LIN {X 783.157, Y -400.206, Z 104.35, A 0, B 90, C -0, E1 0, E2 0, E3 0, E4 0} C_DIS
LIN {X 784.381, Y -394.324, Z 104.35, A 0, B 90, C -0, E1 0, E2 0, E3 0, E4 0} C_DIS
LIN {X 784.236, Y -393.182, Z 104.35, A 0, B 90, C -0, E1 0, E2 0, E3 0, E4 0} C_DIS
LIN {X 783.116, Y -392.84, Z 104.35, A 0, B 90, C -0, E1 0, E2 0, E3 0, E4 0} C_DIS
LIN {X 777.125, Y -392.381, Z 104.35, A 0, B 90, C -0, E1 0, E2 0, E3 0, E4 0} C_DIS
LIN {X 776.023, Y -391.959, Z 104.35, A 0, B 90, C -0, E1 0, E2 0, E3 0, E4 0} C_DIS
LIN {X 775.424, Y -390.936, Z 104.35, A 0, B 90, C -0, E1 0, E2 0, E3 0, E4 0} C_DIS
LIN {X 773.544, Y -385.23, Z 104.35, A 0, B 90, C -0, E1 0, E2 0, E3 0, E4 0} C_DIS
LIN {X 772.847, Y -384.313, Z 104.35, A 0, B 90, C -0, E1 0, E2 0, E3 0, E4 0} C_DIS
LIN {X 771.706, Y -384.577, Z 104.35, A 0, B 90, C -0, E1 0, E2 0, E3 0, E4 0} C_DIS
LIN {X 767.372, Y -386.655, Z 104.35, A 0, B 90, C -0, E1 0, E2 0, E3 0, E4 0} C_DIS
LIN {X 766.095, Y -387.238, Z 105, A 0, B 90, C -0, E1 0, E2 0, E3 0, E4 0} C_DIS
LIN {X 764.935, Y -387.432, Z 105, A 0, B 90, C -0, E1 0, E2 0, E3 0, E4 0} C_DIS
LIN {X 763.905, Y -386.856, Z 105, A 0, B 90, C -0, E1 0, E2 0, E3 0, E4 0} C_DIS
LIN {X 759.412, Y -382.906, Z 105, A 0, B 90, C -0, E1 0, E2 0, E3 0, E4 0} C_DIS
LIN {X 758.351, Y -382.471, Z 105, A 0, B 90, C -0, E1 0, E2 0, E3 0, E4 0} C_DIS
LIN {X 757.504, Y -383.273, Z 105, A 0, B 90, C -0, E1 0, E2 0, E3 0, E4 0} C_DIS
LIN {X 754.164, Y -388.237, Z 105, A 0, B 90, C -0, E1 0, E2 0, E3 0, E4 0} C_DIS
LIN {X 753.257, Y -388.984, Z 105, A 0, B 90, C -0, E1 0, E2 0, E3 0, E4 0} C_DIS
LIN {X 752.077, Y -389, Z 105, A 0, B 90, C -0, E1 0, E2 0, E3 0, E4 0} C_DIS
LIN {X 746.211, Y -387.826, Z 105, A 0, B 90, C -0, E1 0, E2 0, E3 0, E4 0} C_DIS
LIN {X 745.074, Y -387.98, Z 105, A 0, B 90, C -0, E1 0, E2 0, E3 0, E4 0} C_DIS
LIN {X 744.742, Y -389.098, Z 105, A 0, B 90, C -0, E1 0, E2 0, E3 0, E4 0} C_DIS
LIN {X 744.331, Y -395.067, Z 105, A 0, B 90, C -0, E1 0, E2 0, E3 0, E4 0} C_DIS
LIN {X 743.919, Y -396.168, Z 105, A 0, B 90, C -0, E1 0, E2 0, E3 0, E4 0} C_DIS
LIN {X 742.906, Y -396.772, Z 105, A 0, B 90, C -0, E1 0, E2 0, E3 0, E4 0} C_DIS
LIN {X 737.238, Y -398.688, Z 105, A 0, B 90, C -0, E1 0, E2 0, E3 0, E4 0} C_DIS
LIN {X 736.331, Y -399.389, Z 105, A 0, B 90, C -0, E1 0, E2 0, E3 0, E4 0} C_DIS
LIN {X 736.602, Y -400.524, Z 105, A 0, B 90, C -0, E1 0, E2 0, E3 0, E4 0} C_DIS
LIN {X 739.231, Y -405.898, Z 105, A 0, B 90, C -0, E1 0, E2 0, E3 0, E4 0} C_DIS
LIN {X 739.424, Y -407.058, Z 105, A 0, B 90, C -0, E1 0, E2 0, E3 0, E4 0} C_DIS
LIN {X 738.849, Y -408.087, Z 105, A 0, B 90, C -0, E1 0, E2 0, E3 0, E4 0} C_DIS
LIN {X 734.899, Y -412.58, Z 105, A 0, B 90, C -0, E1 0, E2 0, E3 0, E4 0} C_DIS
LIN {X 734.463, Y -413.642, Z 105, A 0, B 90, C -0, E1 0, E2 0, E3 0, E4 0} C_DIS
LIN {X 735.266, Y -414.488, Z 105, A 0, B 90, C -0, E1 0, E2 0, E3 0, E4 0} C_DIS
LIN {X 740.229, Y -417.828, Z 105, A 0, B 90, C -0, E1 0, E2 0, E3 0, E4 0} C_DIS
LIN {X 740.977, Y -418.736, Z 105, A 0, B 90, C -0, E1 0, E2 0, E3 0, E4 0} C_DIS
LIN {X 740.993, Y -419.915, Z 105, A 0, B 90, C -0, E1 0, E2 0, E3 0, E4 0} C_DIS
LIN {X 739.819, Y -425.782, Z 105, A 0, B 90, C -0, E1 0, E2 0, E3 0, E4 0} C_DIS
LIN {X 739.972, Y -426.918, Z 105, A 0, B 90, C -0, E1 0, E2 0, E3 0, E4 0} C_DIS
LIN {X 741.091, Y -427.251, Z 105, A 0, B 90, C -0, E1 0, E2 0, E3 0, E4 0} C_DIS
LIN {X 747.059, Y -427.661, Z 105, A 0, B 90, C -0, E1 0, E2 0, E3 0, E4 0} C_DIS
LIN {X 748.16, Y -428.073, Z 105, A 0, B 90, C -0, E1 0, E2 0, E3 0, E4 0} C_DIS
LIN {X 748.764, Y -429.087, Z 105, A 0, B 90, C -0, E1 0, E2 0, E3 0, E4 0} C_DIS
LIN {X 750.68, Y -434.754, Z 105, A 0, B 90, C -0, E1 0, E2 0, E3 0, E4 0} C_DIS
LIN {X 751.382, Y -435.662, Z 105, A 0, B 90, C -0, E1 0, E2 0, E3 0, E4 0} C_DIS
LIN {X 752.516, Y -435.39, Z 105, A 0, B 90, C -0, E1 0, E2 0, E3 0, E4 0} C_DIS
LIN {X 757.89, Y -432.762, Z 105, A 0, B 90, C -0, E1 0, E2 0, E3 0, E4 0} C_DIS
LIN {X 759.05, Y -432.568, Z 105, A 0, B 90, C -0, E1 0, E2 0, E3 0, E4 0} C_DIS
LIN {X 760.08, Y -433.144, Z 105, A 0, B 90, C -0, E1 0, E2 0, E3 0, E4 0} C_DIS
LIN {X 764.573, Y -437.094, Z 105, A 0, B 90, C -0, E1 0, E2 0, E3 0, E4 0} C_DIS
LIN {X 765.634, Y -437.529, Z 105, A 0, B 90, C -0, E1 0, E2 0, E3 0, E4 0} C_DIS
LIN {X 766.481, Y -436.727, Z 105, A 0, B 90, C -0, E1 0, E2 0, E3 0, E4 0} C_DIS
LIN {X 769.821, Y -431.763, Z 105, A 0, B 90, C -0, E1 0, E2 0, E3 0, E4 0} C_DIS
LIN {X 770.728, Y -431.016, Z 105, A 0, B 90, C -0, E1 0, E2 0, E3 0, E4 0} C_DIS
LIN {X 771.908, Y -431, Z 105, A 0, B 90, C -0, E1 0, E2 0, E3 0, E4 0} C_DIS
LIN {X 777.774, Y -432.174, Z 105, A 0, B 90, C -0, E1 0, E2 0, E3 0, E4 0} C_DIS
LIN {X 778.911, Y -432.02, Z 105, A 0, B 90, C -0, E1 0, E2 0, E3 0, E4 0} C_DIS
LIN {X 779.243, Y -430.902, Z 105, A 0, B 90, C -0, E1 0, E2 0, E3 0, E4 0} C_DIS
LIN {X 779.654, Y -424.933, Z 105, A 0, B 90, C -0, E1 0, E2 0, E3 0, E4 0} C_DIS
LIN {X 780.066, Y -423.832, Z 105, A 0, B 90, C -0, E1 0, E2 0, E3 0, E4 0} C_DIS
LIN {X 781.079, Y -423.228, Z 105, A 0, B 90, C -0, E1 0, E2 0, E3 0, E4 0} C_DIS
LIN {X 786.747, Y -421.312, Z 105, A 0, B 90, C -0, E1 0, E2 0, E3 0, E4 0} C_DIS
LIN {X 787.654, Y -420.611, Z 105, A 0, B 90, C -0, E1 0, E2 0, E3 0, E4 0} C_DIS
LIN {X 787.383, Y -419.476, Z 105, A 0, B 90, C -0, E1 0, E2 0, E3 0, E4 0} C_DIS
LIN {X 784.754, Y -414.102, Z 105, A 0, B 90, C -0, E1 0, E2 0, E3 0, E4 0} C_DIS
LIN {X 784.561, Y -412.942, Z 105, A 0, B 90, C -0, E1 0, E2 0, E3 0, E4 0} C_DIS
LIN {X 785.136, Y -411.913, Z 105, A 0, B 90, C -0, E1 0, E2 0, E3 0, E4 0} C_DIS
LIN {X 789.086, Y -407.42, Z 105, A 0, B 90, C -0, E1 0, E2 0, E3 0, E4 0} C_DIS
LIN {X 789.522, Y -406.358, Z 105, A 0, B 90, C -0, E1 0, E2 0, E3 0, E4 0} C_DIS
LIN {X 788.719, Y -405.512, Z 105, A 0, B 90, C -0, E1 0, E2 0, E3 0, E4 0} C_DIS
LIN {X 783.756, Y -402.172, Z 105, A 0, B 90, C -0, E1 0, E2 0, E3 0, E4 0} C_DIS
LIN {X 783.008, Y -401.264, Z 105, A 0, B 90, C -0, E1 0, E2 0, E3 0, E4 0} C_DIS
LIN {X 782.992, Y -400.085, Z 105, A 0, B 90, C -0, E1 0, E2 0, E3 0, E4 0} C_DIS
LIN {X 784.166, Y -394.218, Z 105, A 0, B 90, C -0, E1 0, E2 0, E3 0, E4 0} C_DIS
LIN {X 784.013, Y -393.082, Z 105, A 0, B 90, C -0, E1 0, E2 0, E3 0, E4 0} C_DIS
LIN {X 782.894, Y -392.749, Z 105, A 0, B 90, C -0, E1 0, E2 0, E3 0, E4 0} C_DIS
LIN {X 776.926, Y -392.339, Z 105, A 0, B 90, C -0, E1 0, E2 0, E3 0, E4 0} C_DIS
LIN {X 775.825, Y -391.927, Z 105, A 0, B 90, C -0, E1 0, E2 0, E3 0, E4 0} C_DIS
LIN {X 775.221, Y -390.913, Z 105, A 0, B 90, C -0, E1 0, E2 0, E3 0, E4 0} C_DIS
LIN {X 773.305, Y -385.246, Z 105, A 0, B 90, C -0, E1 0, E2 0, E3 0, E4 0} C_DIS
LIN {X 772.603, Y -384.338, Z 105, A 0, B 90, C -0, E1 0, E2 0, E3 0, E4 0} C_DIS
LIN {X 771.469, Y -384.61, Z 105, A 0, B 90, C -0, E1 0, E2 0, E3 0, E4 0} C_DIS
LIN {X 767.169, Y -386.712, Z 105, A 0, B 90, C -0, E1 0, E2 0, E3 0, E4 0} C_DIS
LIN {X 765.903, Y -387.302, Z 105.65, A 0, B 90, C -0, E1 0, E2 0, E3 0, E4 0} C_DIS
LIN {X 764.75, Y -387.504, Z 105.65, A 0, B 90, C -0, E1 0, E2 0, E3 0, E4 0} C_DIS
LIN {X 763.72, Y -386.938, Z 105.65, A 0, B 90, C -0, E1 0, E2 0, E3 0, E4 0} C_DIS
LIN {X 759.215, Y -383.039, Z 105.65, A 0, B 90, C -0, E1 0, E2 0, E3 0, E4 0} C_DIS
LIN {X 758.155, Y -382.613, Z 105.65, A 0, B 90, C -0, E1 0, E2 0, E3 0, E4 0} C_DIS
LIN {X 757.318, Y -383.419, Z 105.65, A 0, B 90, C -0, E1 0, E2 0, E3 0, E4 0} C_DIS
LIN {X 754.03, Y -388.387, Z 105.65, A 0, B 90, C -0, E1 0, E2 0, E3 0, E4 0} C_DIS
LIN {X 753.132, Y -389.139, Z 105.65, A 0, B 90, C -0, E1 0, E2 0, E3 0, E4 0} C_DIS
LIN {X 751.958, Y -389.164, Z 105.65, A 0, B 90, C -0, E1 0, E2 0, E3 0, E4 0} C_DIS
LIN {X 746.107, Y -388.04, Z 105.65, A 0, B 90, C -0, E1 0, E2 0, E3 0, E4 0} C_DIS
LIN {X 744.976, Y -388.201, Z 105.65, A 0, B 90, C -0, E1 0, E2 0, E3 0, E4 0} C_DIS
LIN {X 744.654, Y -389.317, Z 105.65, A 0, B 90, C -0, E1 0, E2 0, E3 0, E4 0} C_DIS
LIN {X 744.29, Y -395.264, Z 105.65, A 0, B 90, C -0, E1 0, E2 0, E3 0, E4 0} C_DIS
LIN {X 743.889, Y -396.364, Z 105.65, A 0, B 90, C -0, E1 0, E2 0, E3 0, E4 0} C_DIS
LIN {X 742.884, Y -396.973, Z 105.65, A 0, B 90, C -0, E1 0, E2 0, E3 0, E4 0} C_DIS
LIN {X 737.255, Y -398.924, Z 105.65, A 0, B 90, C -0, E1 0, E2 0, E3 0, E4 0} C_DIS
LIN {X 736.356, Y -399.63, Z 105.65, A 0, B 90, C -0, E1 0, E2 0, E3 0, E4 0} C_DIS
LIN {X 736.635, Y -400.758, Z 105.65, A 0, B 90, C -0, E1 0, E2 0, E3 0, E4 0} C_DIS
LIN {X 739.294, Y -406.089, Z 105.65, A 0, B 90, C -0, E1 0, E2 0, E3 0, E4 0} C_DIS
LIN {X 739.496, Y -407.243, Z 105.65, A 0, B 90, C -0, E1 0, E2 0, E3 0, E4 0} C_DIS
LIN {X 738.93, Y -408.272, Z 105.65, A 0, B 90, C -0, E1 0, E2 0, E3 0, E4 0} C_DIS
LIN {X 735.031, Y -412.777, Z 105.65, A 0, B 90, C -0, E1 0, E2 0, E3 0, E4 0} C_DIS
LIN {X 734.606, Y -413.837, Z 105.65, A 0, B 90, C -0, E1 0, E2 0, E3 0, E4 0} C_DIS
LIN {X 735.411, Y -414.674, Z 105.65, A 0, B 90, C -0, E1 0, E2 0, E3 0, E4 0} C_DIS
LIN {X 740.38, Y -417.962, Z 105.65, A 0, B 90, C -0, E1 0, E2 0, E3 0, E4 0} C_DIS
LIN {X 741.131, Y -418.86, Z 105.65, A 0, B 90, C -0, E1 0, E2 0, E3 0, E4 0} C_DIS
LIN {X 741.156, Y -420.035, Z 105.65, A 0, B 90, C -0, E1 0, E2 0, E3 0, E4 0} C_DIS
LIN {X 740.032, Y -425.886, Z 105.65, A 0, B 90, C -0, E1 0, E2 0, E3 0, E4 0} C_DIS
LIN {X 740.193, Y -427.016, Z 105.65, A 0, B 90, C -0, E1 0, E2 0, E3 0, E4 0} C_DIS
LIN {X 741.31, Y -427.339, Z 105.65, A 0, B 90, C -0, E1 0, E2 0, E3 0, E4 0} C_DIS
LIN {X 747.256, Y -427.702, Z 105.65, A 0, B 90, C -0, E1 0, E2 0, E3 0, E4 0} C_DIS
LIN {X 748.356, Y -428.104, Z 105.65, A 0, B 90, C -0, E1 0, E2 0, E3 0, E4 0} C_DIS
LIN {X 748.965, Y -429.109, Z 105.65, A 0, B 90, C -0, E1 0, E2 0, E3 0, E4 0} C_DIS
LIN {X 750.917, Y -434.738, Z 105.65, A 0, B 90, C -0, E1 0, E2 0, E3 0, E4 0} C_DIS
LIN {X 751.622, Y -435.636, Z 105.65, A 0, B 90, C -0, E1 0, E2 0, E3 0, E4 0} C_DIS
LIN {X 752.75, Y -435.357, Z 105.65, A 0, B 90, C -0, E1 0, E2 0, E3 0, E4 0} C_DIS
LIN {X 758.082, Y -432.698, Z 105.65, A 0, B 90, C -0, E1 0, E2 0, E3 0, E4 0} C_DIS
LIN {X 759.235, Y -432.496, Z 105.65, A 0, B 90, C -0, E1 0, E2 0, E3 0, E4 0} C_DIS
LIN {X 760.265, Y -433.062, Z 105.65, A 0, B 90, C -0, E1 0, E2 0, E3 0, E4 0} C_DIS
LIN {X 764.77, Y -436.961, Z 105.65, A 0, B 90, C -0, E1 0, E2 0, E3 0, E4 0} C_DIS
LIN {X 765.83, Y -437.387, Z 105.65, A 0, B 90, C -0, E1 0, E2 0, E3 0, E4 0} C_DIS
LIN {X 766.667, Y -436.581, Z 105.65, A 0, B 90, C -0, E1 0, E2 0, E3 0, E4 0} C_DIS
LIN {X 769.955, Y -431.613, Z 105.65, A 0, B 90, C -0, E1 0, E2 0, E3 0, E4 0} C_DIS
LIN {X 770.853, Y -430.861, Z 105.65, A 0, B 90, C -0, E1 0, E2 0, E3 0, E4 0} C_DIS
LIN {X 772.027, Y -430.836, Z 105.65, A 0, B 90, C -0, E1 0, E2 0, E3 0, E4 0} C_DIS
LIN {X 777.878, Y -431.96, Z 105.65, A 0, B 90, C -0, E1 0, E2 0, E3 0, E4 0} C_DIS
LIN {X 779.009, Y -431.799, Z 105.65, A 0, B 90, C -0, E1 0, E2 0, E3 0, E4 0} C_DIS
LIN {X 779.331, Y -430.683, Z 105.65, A 0, B 90, C -0, E1 0, E2 0, E3 0, E4 0} C_DIS
LIN {X 779.695, Y -424.736, Z 105.65, A 0, B 90, C -0, E1 0, E2 0, E3 0, E4 0} C_DIS
LIN {X 780.096, Y -423.636, Z 105.65, A 0, B 90, C -0, E1 0, E2 0, E3 0, E4 0} C_DIS
LIN {X 781.101, Y -423.027, Z 105.65, A 0, B 90, C -0, E1 0, E2 0, E3 0, E4 0} C_DIS
LIN {X 786.73, Y -421.076, Z 105.65, A 0, B 90, C -0, E1 0, E2 0, E3 0, E4 0} C_DIS
LIN {X 787.629, Y -420.37, Z 105.65, A 0, B 90, C -0, E1 0, E2 0, E3 0, E4 0} C_DIS
LIN {X 787.349, Y -419.242, Z 105.65, A 0, B 90, C -0, E1 0, E2 0, E3 0, E4 0} C_DIS
LIN {X 784.691, Y -413.911, Z 105.65, A 0, B 90, C -0, E1 0, E2 0, E3 0, E4 0} C_DIS
LIN {X 784.489, Y -412.757, Z 105.65, A 0, B 90, C -0, E1 0, E2 0, E3 0, E4 0} C_DIS
LIN {X 785.055, Y -411.728, Z 105.65, A 0, B 90, C -0, E1 0, E2 0, E3 0, E4 0} C_DIS
LIN {X 788.954, Y -407.223, Z 105.65, A 0, B 90, C -0, E1 0, E2 0, E3 0, E4 0} C_DIS
LIN {X 789.379, Y -406.163, Z 105.65, A 0, B 90, C -0, E1 0, E2 0, E3 0, E4 0} C_DIS
LIN {X 788.573, Y -405.326, Z 105.65, A 0, B 90, C -0, E1 0, E2 0, E3 0, E4 0} C_DIS
LIN {X 783.605, Y -402.038, Z 105.65, A 0, B 90, C -0, E1 0, E2 0, E3 0, E4 0} C_DIS
LIN {X 782.854, Y -401.14, Z 105.65, A 0, B 90, C -0, E1 0, E2 0, E3 0, E4 0} C_DIS
LIN {X 782.829, Y -399.965, Z 105.65, A 0, B 90, C -0, E1 0, E2 0, E3 0, E4 0} C_DIS
LIN {X 783.953, Y -394.114, Z 105.65, A 0, B 90, C -0, E1 0, E2 0, E3 0, E4 0} C_DIS
LIN {X 783.791, Y -392.984, Z 105.65, A 0, B 90, C -0, E1 0, E2 0, E3 0, E4 0} C_DIS
LIN {X 782.675, Y -392.661, Z 105.65, A 0, B 90, C -0, E1 0, E2 0, E3 0, E4 0} C_DIS
LIN {X 776.728, Y -392.298, Z 105.65, A 0, B 90, C -0, E1 0, E2 0, E3 0, E4 0} C_DIS
LIN {X 775.629, Y -391.896, Z 105.65, A 0, B 90, C -0, E1 0, E2 0, E3 0, E4 0} C_DIS
LIN {X 775.02, Y -390.891, Z 105.65, A 0, B 90, C -0, E1 0, E2 0, E3 0, E4 0} C_DIS
LIN {X 773.068, Y -385.262, Z 105.65, A 0, B 90, C -0, E1 0, E2 0, E3 0, E4 0} C_DIS
LIN {X 772.363, Y -384.364, Z 105.65, A 0, B 90, C -0, E1 0, E2 0, E3 0, E4 0} C_DIS
LIN {X 771.235, Y -384.643, Z 105.65, A 0, B 90, C -0, E1 0, E2 0, E3 0, E4 0} C_DIS
LIN {X 766.97, Y -386.77, Z 105.65, A 0, B 90, C -0, E1 0, E2 0, E3 0, E4 0} C_DIS
LIN {X 765.714, Y -387.365, Z 106.3, A 0, B 90, C -0, E1 0, E2 0, E3 0, E4 0} C_DIS
LIN {X 764.567, Y -387.575, Z 106.3, A 0, B 90, C -0, E1 0, E2 0, E3 0, E4 0} C_DIS
LIN {X 763.537, Y -387.02, Z 106.3, A 0, B 90, C -0, E1 0, E2 0, E3 0, E4 0} C_DIS
LIN {X 759.022, Y -383.171, Z 106.3, A 0, B 90, C -0, E1 0, E2 0, E3 0, E4 0} C_DIS
LIN {X 757.963, Y -382.755, Z 106.3, A 0, B 90, C -0, E1 0, E2 0, E3 0, E4 0} C_DIS
LIN {X 757.135, Y -383.564, Z 106.3, A 0, B 90, C -0, E1 0, E2 0, E3 0, E4 0} C_DIS
LIN {X 753.898, Y -388.537, Z 106.3, A 0, B 90, C -0, E1 0, E2 0, E3 0, E4 0} C_DIS
LIN {X 753.01, Y -389.292, Z 106.3, A 0, B 90, C -0, E1 0, E2 0, E3 0, E4 0} C_DIS
LIN {X 751.84, Y -389.326, Z 106.3, A 0, B 90, C -0, E1 0, E2 0, E3 0, E4 0} C_DIS
LIN {X 746.005, Y -388.251, Z 106.3, A 0, B 90, C -0, E1 0, E2 0, E3 0, E4 0} C_DIS
LIN {X 744.88, Y -388.42, Z 106.3, A 0, B 90, C -0, E1 0, E2 0, E3 0, E4 0} C_DIS
LIN {X 744.568, Y -389.534, Z 106.3, A 0, B 90, C -0, E1 0, E2 0, E3 0, E4 0} C_DIS
LIN {X 744.251, Y -395.459, Z 106.3, A 0, B 90, C -0, E1 0, E2 0, E3 0, E4 0} C_DIS
LIN {X 743.859, Y -396.558, Z 106.3, A 0, B 90, C -0, E1 0, E2 0, E3 0, E4 0} C_DIS
LIN {X 742.864, Y -397.172, Z 106.3, A 0, B 90, C -0, E1 0, E2 0, E3 0, E4 0} C_DIS
LIN {X 737.273, Y -399.158, Z 106.3, A 0, B 90, C -0, E1 0, E2 0, E3 0, E4 0} C_DIS
LIN {X 736.383, Y -399.867, Z 106.3, A 0, B 90, C -0, E1 0, E2 0, E3 0, E4 0} C_DIS
LIN {X 736.67, Y -400.989, Z 106.3, A 0, B 90, C -0, E1 0, E2 0, E3 0, E4 0} C_DIS
LIN {X 739.358, Y -406.278, Z 106.3, A 0, B 90, C -0, E1 0, E2 0, E3 0, E4 0} C_DIS
LIN {X 739.568, Y -407.425, Z 106.3, A 0, B 90, C -0, E1 0, E2 0, E3 0, E4 0} C_DIS
LIN {X 739.012, Y -408.455, Z 106.3, A 0, B 90, C -0, E1 0, E2 0, E3 0, E4 0} C_DIS
LIN {X 735.164, Y -412.971, Z 106.3, A 0, B 90, C -0, E1 0, E2 0, E3 0, E4 0} C_DIS
LIN {X 734.748, Y -414.03, Z 106.3, A 0, B 90, C -0, E1 0, E2 0, E3 0, E4 0} C_DIS
LIN {X 735.557, Y -414.857, Z 106.3, A 0, B 90, C -0, E1 0, E2 0, E3 0, E4 0} C_DIS
LIN {X 740.529, Y -418.094, Z 106.3, A 0, B 90, C -0, E1 0, E2 0, E3 0, E4 0} C_DIS
LIN {X 741.285, Y -418.982, Z 106.3, A 0, B 90, C -0, E1 0, E2 0, E3 0, E4 0} C_DIS
LIN {X 741.319, Y -420.152, Z 106.3, A 0, B 90, C -0, E1 0, E2 0, E3 0, E4 0} C_DIS
LIN {X 740.243, Y -425.987, Z 106.3, A 0, B 90, C -0, E1 0, E2 0, E3 0, E4 0} C_DIS
LIN {X 740.413, Y -427.112, Z 106.3, A 0, B 90, C -0, E1 0, E2 0, E3 0, E4 0} C_DIS
LIN {X 741.527, Y -427.425, Z 106.3, A 0, B 90, C -0, E1 0, E2 0, E3 0, E4 0} C_DIS
LIN {X 747.452, Y -427.741, Z 106.3, A 0, B 90, C -0, E1 0, E2 0, E3 0, E4 0} C_DIS
LIN {X 748.55, Y -428.133, Z 106.3, A 0, B 90, C -0, E1 0, E2 0, E3 0, E4 0} C_DIS
LIN {X 749.164, Y -429.129, Z 106.3, A 0, B 90, C -0, E1 0, E2 0, E3 0, E4 0} C_DIS
LIN {X 751.151, Y -434.72, Z 106.3, A 0, B 90, C -0, E1 0, E2 0, E3 0, E4 0} C_DIS
LIN {X 751.86, Y -435.609, Z 106.3, A 0, B 90, C -0, E1 0, E2 0, E3 0, E4 0} C_DIS
LIN {X 752.981, Y -435.323, Z 106.3, A 0, B 90, C -0, E1 0, E2 0, E3 0, E4 0} C_DIS
LIN {X 758.271, Y -432.635, Z 106.3, A 0, B 90, C -0, E1 0, E2 0, E3 0, E4 0} C_DIS
LIN {X 759.418, Y -432.425, Z 106.3, A 0, B 90, C -0, E1 0, E2 0, E3 0, E4 0} C_DIS
LIN {X 760.447, Y -432.98, Z 106.3, A 0, B 90, C -0, E1 0, E2 0, E3 0, E4 0} C_DIS
LIN {X 764.963, Y -436.829, Z 106.3, A 0, B 90, C -0, E1 0, E2 0, E3 0, E4 0} C_DIS
LIN {X 766.022, Y -437.245, Z 106.3, A 0, B 90, C -0, E1 0, E2 0, E3 0, E4 0} C_DIS
LIN {X 766.85, Y -436.436, Z 106.3, A 0, B 90, C -0, E1 0, E2 0, E3 0, E4 0} C_DIS
LIN {X 770.087, Y -431.463, Z 106.3, A 0, B 90, C -0, E1 0, E2 0, E3 0, E4 0} C_DIS
LIN {X 770.975, Y -430.708, Z 106.3, A 0, B 90, C -0, E1 0, E2 0, E3 0, E4 0} C_DIS
LIN {X 772.145, Y -430.674, Z 106.3, A 0, B 90, C -0, E1 0, E2 0, E3 0, E4 0} C_DIS
LIN {X 777.98, Y -431.749, Z 106.3, A 0, B 90, C -0, E1 0, E2 0, E3 0, E4 0} C_DIS
LIN {X 779.105, Y -431.58, Z 106.3, A 0, B 90, C -0, E1 0, E2 0, E3 0, E4 0} C_DIS
LIN {X 779.417, Y -430.466, Z 106.3, A 0, B 90, C -0, E1 0, E2 0, E3 0, E4 0} C_DIS
LIN {X 779.734, Y -424.541, Z 106.3, A 0, B 90, C -0, E1 0, E2 0, E3 0, E4 0} C_DIS
LIN {X 780.125, Y -423.442, Z 106.3, A 0, B 90, C -0, E1 0, E2 0, E3 0, E4 0} C_DIS
LIN {X 781.121, Y -422.828, Z 106.3, A 0, B 90, C -0, E1 0, E2 0, E3 0, E4 0} C_DIS
LIN {X 786.712, Y -420.842, Z 106.3, A 0, B 90, C -0, E1 0, E2 0, E3 0, E4 0} C_DIS
LIN {X 787.602, Y -420.133, Z 106.3, A 0, B 90, C -0, E1 0, E2 0, E3 0, E4 0} C_DIS
LIN {X 787.315, Y -419.011, Z 106.3, A 0, B 90, C -0, E1 0, E2 0, E3 0, E4 0} C_DIS
LIN {X 784.627, Y -413.722, Z 106.3, A 0, B 90, C -0, E1 0, E2 0, E3 0, E4 0} C_DIS
LIN {X 784.417, Y -412.575, Z 106.3, A 0, B 90, C -0, E1 0, E2 0, E3 0, E4 0} C_DIS
LIN {X 784.973, Y -411.545, Z 106.3, A 0, B 90, C -0, E1 0, E2 0, E3 0, E4 0} C_DIS
LIN {X 788.821, Y -407.029, Z 106.3, A 0, B 90, C -0, E1 0, E2 0, E3 0, E4 0} C_DIS
LIN {X 789.237, Y -405.97, Z 106.3, A 0, B 90, C -0, E1 0, E2 0, E3 0, E4 0} C_DIS
LIN {X 788.428, Y -405.143, Z 106.3, A 0, B 90, C -0, E1 0, E2 0, E3 0, E4 0} C_DIS
LIN {X 783.456, Y -401.906, Z 106.3, A 0, B 90, C -0, E1 0, E2 0, E3 0, E4 0} C_DIS
LIN {X 782.7, Y -401.018, Z 106.3, A 0, B 90, C -0, E1 0, E2 0, E3 0, E4 0} C_DIS
LIN {X 782.666, Y -399.848, Z 106.3, A 0, B 90, C -0, E1 0, E2 0, E3 0, E4 0} C_DIS
LIN {X 783.742, Y -394.013, Z 106.3, A 0, B 90, C -0, E1 0, E2 0, E3 0, E4 0} C_DIS
LIN {X 783.572, Y -392.888, Z 106.3, A 0, B 90, C -0, E1 0, E2 0, E3 0, E4 0} C_DIS
LIN {X 782.458, Y -392.575, Z 106.3, A 0, B 90, C -0, E1 0, E2 0, E3 0, E4 0} C_DIS
LIN {X 776.533, Y -392.259, Z 106.3, A 0, B 90, C -0, E1 0, E2 0, E3 0, E4 0} C_DIS
LIN {X 775.435, Y -391.867, Z 106.3, A 0, B 90, C -0, E1 0, E2 0, E3 0, E4 0} C_DIS
LIN {X 774.821, Y -390.871, Z 106.3, A 0, B 90, C -0, E1 0, E2 0, E3 0, E4 0} C_DIS
LIN {X 772.834, Y -385.28, Z 106.3, A 0, B 90, C -0, E1 0, E2 0, E3 0, E4 0} C_DIS
LIN {X 772.125, Y -384.391, Z 106.3, A 0, B 90, C -0, E1 0, E2 0, E3 0, E4 0} C_DIS
LIN {X 771.004, Y -384.677, Z 106.3, A 0, B 90, C -0, E1 0, E2 0, E3 0, E4 0} C_DIS
LIN {X 766.772, Y -386.828, Z 106.3, A 0, B 90, C -0, E1 0, E2 0, E3 0, E4 0} C_DIS
LIN {X 765.528, Y -387.429, Z 106.95, A 0, B 90, C -0, E1 0, E2 0, E3 0, E4 0} C_DIS
LIN {X 764.387, Y -387.647, Z 106.95, A 0, B 90, C -0, E1 0, E2 0, E3 0, E4 0} C_DIS
LIN {X 763.357, Y -387.102, Z 106.95, A 0, B 90, C -0, E1 0, E2 0, E3 0, E4 0} C_DIS
LIN {X 758.831, Y -383.303, Z 106.95, A 0, B 90, C -0, E1 0, E2 0, E3 0, E4 0} C_DIS
LIN {X 757.773, Y -382.897, Z 106.95, A 0, B 90, C -0, E1 0, E2 0, E3 0, E4 0} C_DIS
LIN {X 756.955, Y -383.708, Z 106.95, A 0, B 90, C -0, E1 0, E2 0, E3 0, E4 0} C_DIS
LIN {X 753.769, Y -388.685, Z 106.95, A 0, B 90, C -0, E1 0, E2 0, E3 0, E4 0} C_DIS
LIN {X 752.89, Y -389.444, Z 106.95, A 0, B 90, C -0, E1 0, E2 0, E3 0, E4 0} C_DIS
LIN {X 751.725, Y -389.487, Z 106.95, A 0, B 90, C -0, E1 0, E2 0, E3 0, E4 0} C_DIS
LIN {X 745.906, Y -388.46, Z 106.95, A 0, B 90, C -0, E1 0, E2 0, E3 0, E4 0} C_DIS
LIN {X 744.787, Y -388.637, Z 106.95, A 0, B 90, C -0, E1 0, E2 0, E3 0, E4 0} C_DIS
LIN {X 744.484, Y -389.749, Z 106.95, A 0, B 90, C -0, E1 0, E2 0, E3 0, E4 0} C_DIS
LIN {X 744.213, Y -395.653, Z 106.95, A 0, B 90, C -0, E1 0, E2 0, E3 0, E4 0} C_DIS
LIN {X 743.832, Y -396.749, Z 106.95, A 0, B 90, C -0, E1 0, E2 0, E3 0, E4 0} C_DIS
LIN {X 742.844, Y -397.369, Z 106.95, A 0, B 90, C -0, E1 0, E2 0, E3 0, E4 0} C_DIS
LIN {X 737.291, Y -399.389, Z 106.95, A 0, B 90, C -0, E1 0, E2 0, E3 0, E4 0} C_DIS
LIN {X 736.411, Y -400.102, Z 106.95, A 0, B 90, C -0, E1 0, E2 0, E3 0, E4 0} C_DIS
LIN {X 736.704, Y -401.217, Z 106.95, A 0, B 90, C -0, E1 0, E2 0, E3 0, E4 0} C_DIS
LIN {X 739.422, Y -406.464, Z 106.95, A 0, B 90, C -0, E1 0, E2 0, E3 0, E4 0} C_DIS
LIN {X 739.639, Y -407.605, Z 106.95, A 0, B 90, C -0, E1 0, E2 0, E3 0, E4 0} C_DIS
LIN {X 739.094, Y -408.635, Z 106.95, A 0, B 90, C -0, E1 0, E2 0, E3 0, E4 0} C_DIS
LIN {X 735.295, Y -413.162, Z 106.95, A 0, B 90, C -0, E1 0, E2 0, E3 0, E4 0} C_DIS
LIN {X 734.889, Y -414.219, Z 106.95, A 0, B 90, C -0, E1 0, E2 0, E3 0, E4 0} C_DIS
LIN {X 735.701, Y -415.038, Z 106.95, A 0, B 90, C -0, E1 0, E2 0, E3 0, E4 0} C_DIS
LIN {X 740.678, Y -418.224, Z 106.95, A 0, B 90, C -0, E1 0, E2 0, E3 0, E4 0} C_DIS
LIN {X 741.437, Y -419.103, Z 106.95, A 0, B 90, C -0, E1 0, E2 0, E3 0, E4 0} C_DIS
LIN {X 741.479, Y -420.267, Z 106.95, A 0, B 90, C -0, E1 0, E2 0, E3 0, E4 0} C_DIS
LIN {X 740.453, Y -426.087, Z 106.95, A 0, B 90, C -0, E1 0, E2 0, E3 0, E4 0} C_DIS
LIN {X 740.63, Y -427.206, Z 106.95, A 0, B 90, C -0, E1 0, E2 0, E3 0, E4 0} C_DIS
LIN {X 741.742, Y -427.509, Z 106.95, A 0, B 90, C -0, E1 0, E2 0, E3 0, E4 0} C_DIS
LIN {X 747.645, Y -427.779, Z 106.95, A 0, B 90, C -0, E1 0, E2 0, E3 0, E4 0} C_DIS
LIN {X 748.742, Y -428.161, Z 106.95, A 0, B 90, C -0, E1 0, E2 0, E3 0, E4 0} C_DIS
LIN {X 749.361, Y -429.148, Z 106.95, A 0, B 90, C -0, E1 0, E2 0, E3 0, E4 0} C_DIS
LIN {X 751.382, Y -434.701, Z 106.95, A 0, B 90, C -0, E1 0, E2 0, E3 0, E4 0} C_DIS
LIN {X 752.095, Y -435.582, Z 106.95, A 0, B 90, C -0, E1 0, E2 0, E3 0, E4 0} C_DIS
LIN {X 753.209, Y -435.288, Z 106.95, A 0, B 90, C -0, E1 0, E2 0, E3 0, E4 0} C_DIS
LIN {X 758.457, Y -432.571, Z 106.95, A 0, B 90, C -0, E1 0, E2 0, E3 0, E4 0} C_DIS
LIN {X 759.598, Y -432.353, Z 106.95, A 0, B 90, C -0, E1 0, E2 0, E3 0, E4 0} C_DIS
LIN {X 760.628, Y -432.898, Z 106.95, A 0, B 90, C -0, E1 0, E2 0, E3 0, E4 0} C_DIS
LIN {X 765.154, Y -436.697, Z 106.95, A 0, B 90, C -0, E1 0, E2 0, E3 0, E4 0} C_DIS
LIN {X 766.212, Y -437.103, Z 106.95, A 0, B 90, C -0, E1 0, E2 0, E3 0, E4 0} C_DIS
LIN {X 767.03, Y -436.292, Z 106.95, A 0, B 90, C -0, E1 0, E2 0, E3 0, E4 0} C_DIS
LIN {X 770.216, Y -431.315, Z 106.95, A 0, B 90, C -0, E1 0, E2 0, E3 0, E4 0} C_DIS
LIN {X 771.095, Y -430.556, Z 106.95, A 0, B 90, C -0, E1 0, E2 0, E3 0, E4 0} C_DIS
LIN {X 772.26, Y -430.513, Z 106.95, A 0, B 90, C -0, E1 0, E2 0, E3 0, E4 0} C_DIS
LIN {X 778.079, Y -431.54, Z 106.95, A 0, B 90, C -0, E1 0, E2 0, E3 0, E4 0} C_DIS
LIN {X 779.198, Y -431.363, Z 106.95, A 0, B 90, C -0, E1 0, E2 0, E3 0, E4 0} C_DIS
LIN {X 779.501, Y -430.251, Z 106.95, A 0, B 90, C -0, E1 0, E2 0, E3 0, E4 0} C_DIS
LIN {X 779.772, Y -424.347, Z 106.95, A 0, B 90, C -0, E1 0, E2 0, E3 0, E4 0} C_DIS
LIN {X 780.153, Y -423.251, Z 106.95, A 0, B 90, C -0, E1 0, E2 0, E3 0, E4 0} C_DIS
LIN {X 781.141, Y -422.631, Z 106.95, A 0, B 90, C -0, E1 0, E2 0, E3 0, E4 0} C_DIS
LIN {X 786.694, Y -420.611, Z 106.95, A 0, B 90, C -0, E1 0, E2 0, E3 0, E4 0} C_DIS
LIN {X 787.574, Y -419.898, Z 106.95, A 0, B 90, C -0, E1 0, E2 0, E3 0, E4 0} C_DIS
LIN {X 787.281, Y -418.783, Z 106.95, A 0, B 90, C -0, E1 0, E2 0, E3 0, E4 0} C_DIS
LIN {X 784.563, Y -413.536, Z 106.95, A 0, B 90, C -0, E1 0, E2 0, E3 0, E4 0} C_DIS
LIN {X 784.346, Y -412.395, Z 106.95, A 0, B 90, C -0, E1 0, E2 0, E3 0, E4 0} C_DIS
LIN {X 784.891, Y -411.365, Z 106.95, A 0, B 90, C -0, E1 0, E2 0, E3 0, E4 0} C_DIS
LIN {X 788.69, Y -406.838, Z 106.95, A 0, B 90, C -0, E1 0, E2 0, E3 0, E4 0} C_DIS
LIN {X 789.096, Y -405.781, Z 106.95, A 0, B 90, C -0, E1 0, E2 0, E3 0, E4 0} C_DIS
LIN {X 788.284, Y -404.962, Z 106.95, A 0, B 90, C -0, E1 0, E2 0, E3 0, E4 0} C_DIS
LIN {X 783.307, Y -401.776, Z 106.95, A 0, B 90, C -0, E1 0, E2 0, E3 0, E4 0} C_DIS
LIN {X 782.548, Y -400.897, Z 106.95, A 0, B 90, C -0, E1 0, E2 0, E3 0, E4 0} C_DIS
LIN {X 782.506, Y -399.733, Z 106.95, A 0, B 90, C -0, E1 0, E2 0, E3 0, E4 0} C_DIS
LIN {X 783.532, Y -393.913, Z 106.95, A 0, B 90, C -0, E1 0, E2 0, E3 0, E4 0} C_DIS
LIN {X 783.355, Y -392.794, Z 106.95, A 0, B 90, C -0, E1 0, E2 0, E3 0, E4 0} C_DIS
LIN {X 782.243, Y -392.491, Z 106.95, A 0, B 90, C -0, E1 0, E2 0, E3 0, E4 0} C_DIS
LIN {X 776.34, Y -392.221, Z 106.95, A 0, B 90, C -0, E1 0, E2 0, E3 0, E4 0} C_DIS
LIN {X 775.243, Y -391.839, Z 106.95, A 0, B 90, C -0, E1 0, E2 0, E3 0, E4 0} C_DIS
LIN {X 774.624, Y -390.852, Z 106.95, A 0, B 90, C -0, E1 0, E2 0, E3 0, E4 0} C_DIS
LIN {X 772.603, Y -385.299, Z 106.95, A 0, B 90, C -0, E1 0, E2 0, E3 0, E4 0} C_DIS
LIN {X 771.89, Y -384.418, Z 106.95, A 0, B 90, C -0, E1 0, E2 0, E3 0, E4 0} C_DIS
LIN {X 770.776, Y -384.712, Z 106.95, A 0, B 90, C -0, E1 0, E2 0, E3 0, E4 0} C_DIS
LIN {X 766.578, Y -386.886, Z 106.95, A 0, B 90, C -0, E1 0, E2 0, E3 0, E4 0} C_DIS
LIN {X 765.344, Y -387.493, Z 107.6, A 0, B 90, C -0, E1 0, E2 0, E3 0, E4 0} C_DIS
LIN {X 764.21, Y -387.719, Z 107.6, A 0, B 90, C -0, E1 0, E2 0, E3 0, E4 0} C_DIS
LIN {X 763.18, Y -387.183, Z 107.6, A 0, B 90, C -0, E1 0, E2 0, E3 0, E4 0} C_DIS
LIN {X 758.643, Y -383.434, Z 107.6, A 0, B 90, C -0, E1 0, E2 0, E3 0, E4 0} C_DIS
LIN {X 757.586, Y -383.037, Z 107.6, A 0, B 90, C -0, E1 0, E2 0, E3 0, E4 0} C_DIS
LIN {X 756.778, Y -383.852, Z 107.6, A 0, B 90, C -0, E1 0, E2 0, E3 0, E4 0} C_DIS
LIN {X 753.642, Y -388.833, Z 107.6, A 0, B 90, C -0, E1 0, E2 0, E3 0, E4 0} C_DIS
LIN {X 752.772, Y -389.595, Z 107.6, A 0, B 90, C -0, E1 0, E2 0, E3 0, E4 0} C_DIS
LIN {X 751.612, Y -389.646, Z 107.6, A 0, B 90, C -0, E1 0, E2 0, E3 0, E4 0} C_DIS
LIN {X 745.808, Y -388.668, Z 107.6, A 0, B 90, C -0, E1 0, E2 0, E3 0, E4 0} C_DIS
LIN {X 744.695, Y -388.852, Z 107.6, A 0, B 90, C -0, E1 0, E2 0, E3 0, E4 0} C_DIS
LIN {X 744.402, Y -389.962, Z 107.6, A 0, B 90, C -0, E1 0, E2 0, E3 0, E4 0} C_DIS
LIN {X 744.177, Y -395.844, Z 107.6, A 0, B 90, C -0, E1 0, E2 0, E3 0, E4 0} C_DIS
LIN {X 743.805, Y -396.939, Z 107.6, A 0, B 90, C -0, E1 0, E2 0, E3 0, E4 0} C_DIS
LIN {X 742.826, Y -397.563, Z 107.6, A 0, B 90, C -0, E1 0, E2 0, E3 0, E4 0} C_DIS
LIN {X 737.31, Y -399.618, Z 107.6, A 0, B 90, C -0, E1 0, E2 0, E3 0, E4 0} C_DIS
LIN {X 736.439, Y -400.334, Z 107.6, A 0, B 90, C -0, E1 0, E2 0, E3 0, E4 0} C_DIS
LIN {X 736.74, Y -401.442, Z 107.6, A 0, B 90, C -0, E1 0, E2 0, E3 0, E4 0} C_DIS
LIN {X 739.486, Y -406.648, Z 107.6, A 0, B 90, C -0, E1 0, E2 0, E3 0, E4 0} C_DIS
LIN {X 739.711, Y -407.783, Z 107.6, A 0, B 90, C -0, E1 0, E2 0, E3 0, E4 0} C_DIS
LIN {X 739.176, Y -408.813, Z 107.6, A 0, B 90, C -0, E1 0, E2 0, E3 0, E4 0} C_DIS
LIN {X 735.426, Y -413.35, Z 107.6, A 0, B 90, C -0, E1 0, E2 0, E3 0, E4 0} C_DIS
LIN {X 735.029, Y -414.406, Z 107.6, A 0, B 90, C -0, E1 0, E2 0, E3 0, E4 0} C_DIS
LIN {X 735.844, Y -415.215, Z 107.6, A 0, B 90, C -0, E1 0, E2 0, E3 0, E4 0} C_DIS
LIN {X 740.825, Y -418.351, Z 107.6, A 0, B 90, C -0, E1 0, E2 0, E3 0, E4 0} C_DIS
LIN {X 741.588, Y -419.221, Z 107.6, A 0, B 90, C -0, E1 0, E2 0, E3 0, E4 0} C_DIS
LIN {X 741.639, Y -420.38, Z 107.6, A 0, B 90, C -0, E1 0, E2 0, E3 0, E4 0} C_DIS
LIN {X 740.66, Y -426.184, Z 107.6, A 0, B 90, C -0, E1 0, E2 0, E3 0, E4 0} C_DIS
LIN {X 740.845, Y -427.297, Z 107.6, A 0, B 90, C -0, E1 0, E2 0, E3 0, E4 0} C_DIS
LIN {X 741.955, Y -427.59, Z 107.6, A 0, B 90, C -0, E1 0, E2 0, E3 0, E4 0} C_DIS
LIN {X 747.836, Y -427.816, Z 107.6, A 0, B 90, C -0, E1 0, E2 0, E3 0, E4 0} C_DIS
LIN {X 748.932, Y -428.188, Z 107.6, A 0, B 90, C -0, E1 0, E2 0, E3 0, E4 0} C_DIS
LIN {X 749.556, Y -429.166, Z 107.6, A 0, B 90, C -0, E1 0, E2 0, E3 0, E4 0} C_DIS
LIN {X 751.61, Y -434.682, Z 107.6, A 0, B 90, C -0, E1 0, E2 0, E3 0, E4 0} C_DIS
LIN {X 752.327, Y -435.554, Z 107.6, A 0, B 90, C -0, E1 0, E2 0, E3 0, E4 0} C_DIS
LIN {X 753.435, Y -435.253, Z 107.6, A 0, B 90, C -0, E1 0, E2 0, E3 0, E4 0} C_DIS
LIN {X 758.641, Y -432.507, Z 107.6, A 0, B 90, C -0, E1 0, E2 0, E3 0, E4 0} C_DIS
LIN {X 759.775, Y -432.281, Z 107.6, A 0, B 90, C -0, E1 0, E2 0, E3 0, E4 0} C_DIS
LIN {X 760.805, Y -432.817, Z 107.6, A 0, B 90, C -0, E1 0, E2 0, E3 0, E4 0} C_DIS
LIN {X 765.342, Y -436.566, Z 107.6, A 0, B 90, C -0, E1 0, E2 0, E3 0, E4 0} C_DIS
LIN {X 766.399, Y -436.963, Z 107.6, A 0, B 90, C -0, E1 0, E2 0, E3 0, E4 0} C_DIS
LIN {X 767.207, Y -436.148, Z 107.6, A 0, B 90, C -0, E1 0, E2 0, E3 0, E4 0} C_DIS
LIN {X 770.343, Y -431.167, Z 107.6, A 0, B 90, C -0, E1 0, E2 0, E3 0, E4 0} C_DIS
LIN {X 771.213, Y -430.405, Z 107.6, A 0, B 90, C -0, E1 0, E2 0, E3 0, E4 0} C_DIS
LIN {X 772.373, Y -430.354, Z 107.6, A 0, B 90, C -0, E1 0, E2 0, E3 0, E4 0} C_DIS
LIN {X 778.177, Y -431.332, Z 107.6, A 0, B 90, C -0, E1 0, E2 0, E3 0, E4 0} C_DIS
LIN {X 779.29, Y -431.148, Z 107.6, A 0, B 90, C -0, E1 0, E2 0, E3 0, E4 0} C_DIS
LIN {X 779.583, Y -430.038, Z 107.6, A 0, B 90, C -0, E1 0, E2 0, E3 0, E4 0} C_DIS
LIN {X 779.808, Y -424.156, Z 107.6, A 0, B 90, C -0, E1 0, E2 0, E3 0, E4 0} C_DIS
LIN {X 780.18, Y -423.061, Z 107.6, A 0, B 90, C -0, E1 0, E2 0, E3 0, E4 0} C_DIS
LIN {X 781.159, Y -422.437, Z 107.6, A 0, B 90, C -0, E1 0, E2 0, E3 0, E4 0} C_DIS
LIN {X 786.675, Y -420.382, Z 107.6, A 0, B 90, C -0, E1 0, E2 0, E3 0, E4 0} C_DIS
LIN {X 787.546, Y -419.666, Z 107.6, A 0, B 90, C -0, E1 0, E2 0, E3 0, E4 0} C_DIS
LIN {X 787.245, Y -418.558, Z 107.6, A 0, B 90, C -0, E1 0, E2 0, E3 0, E4 0} C_DIS
LIN {X 784.499, Y -413.352, Z 107.6, A 0, B 90, C -0, E1 0, E2 0, E3 0, E4 0} C_DIS
LIN {X 784.274, Y -412.217, Z 107.6, A 0, B 90, C -0, E1 0, E2 0, E3 0, E4 0} C_DIS
LIN {X 784.809, Y -411.187, Z 107.6, A 0, B 90, C -0, E1 0, E2 0, E3 0, E4 0} C_DIS
LIN {X 788.559, Y -406.65, Z 107.6, A 0, B 90, C -0, E1 0, E2 0, E3 0, E4 0} C_DIS
LIN {X 788.955, Y -405.594, Z 107.6, A 0, B 90, C -0, E1 0, E2 0, E3 0, E4 0} C_DIS
LIN {X 788.141, Y -404.785, Z 107.6, A 0, B 90, C -0, E1 0, E2 0, E3 0, E4 0} C_DIS
LIN {X 783.16, Y -401.649, Z 107.6, A 0, B 90, C -0, E1 0, E2 0, E3 0, E4 0} C_DIS
LIN {X 782.397, Y -400.779, Z 107.6, A 0, B 90, C -0, E1 0, E2 0, E3 0, E4 0} C_DIS
LIN {X 782.346, Y -399.62, Z 107.6, A 0, B 90, C -0, E1 0, E2 0, E3 0, E4 0} C_DIS
LIN {X 783.325, Y -393.816, Z 107.6, A 0, B 90, C -0, E1 0, E2 0, E3 0, E4 0} C_DIS
LIN {X 783.14, Y -392.703, Z 107.6, A 0, B 90, C -0, E1 0, E2 0, E3 0, E4 0} C_DIS
LIN {X 782.03, Y -392.41, Z 107.6, A 0, B 90, C -0, E1 0, E2 0, E3 0, E4 0} C_DIS
LIN {X 776.149, Y -392.184, Z 107.6, A 0, B 90, C -0, E1 0, E2 0, E3 0, E4 0} C_DIS
LIN {X 775.053, Y -391.812, Z 107.6, A 0, B 90, C -0, E1 0, E2 0, E3 0, E4 0} C_DIS
LIN {X 774.429, Y -390.834, Z 107.6, A 0, B 90, C -0, E1 0, E2 0, E3 0, E4 0} C_DIS
LIN {X 772.375, Y -385.318, Z 107.6, A 0, B 90, C -0, E1 0, E2 0, E3 0, E4 0} C_DIS
LIN {X 771.658, Y -384.446, Z 107.6, A 0, B 90, C -0, E1 0, E2 0, E3 0, E4 0} C_DIS
LIN {X 770.55, Y -384.747, Z 107.6, A 0, B 90, C -0, E1 0, E2 0, E3 0, E4 0} C_DIS
LIN {X 766.385, Y -386.944, Z 107.6, A 0, B 90, C -0, E1 0, E2 0, E3 0, E4 0} C_DIS
LIN {X 765.163, Y -387.557, Z 108.25, A 0, B 90, C -0, E1 0, E2 0, E3 0, E4 0} C_DIS
LIN {X 764.035, Y -387.79, Z 108.25, A 0, B 90, C -0, E1 0, E2 0, E3 0, E4 0} C_DIS
LIN {X 763.005, Y -387.265, Z 108.25, A 0, B 90, C -0, E1 0, E2 0, E3 0, E4 0} C_DIS
LIN {X 758.458, Y -383.564, Z 108.25, A 0, B 90, C -0, E1 0, E2 0, E3 0, E4 0} C_DIS
LIN {X 757.402, Y -383.177, Z 108.25, A 0, B 90, C -0, E1 0, E2 0, E3 0, E4 0} C_DIS
LIN {X 756.603, Y -383.994, Z 108.25, A 0, B 90, C -0, E1 0, E2 0, E3 0, E4 0} C_DIS
LIN {X 753.517, Y -388.979, Z 108.25, A 0, B 90, C -0, E1 0, E2 0, E3 0, E4 0} C_DIS
LIN {X 752.656, Y -389.745, Z 108.25, A 0, B 90, C -0, E1 0, E2 0, E3 0, E4 0} C_DIS
LIN {X 751.501, Y -389.804, Z 108.25, A 0, B 90, C -0, E1 0, E2 0, E3 0, E4 0} C_DIS
LIN {X 745.713, Y -388.873, Z 108.25, A 0, B 90, C -0, E1 0, E2 0, E3 0, E4 0} C_DIS
LIN {X 744.606, Y -389.065, Z 108.25, A 0, B 90, C -0, E1 0, E2 0, E3 0, E4 0} C_DIS
LIN {X 744.322, Y -390.173, Z 108.25, A 0, B 90, C -0, E1 0, E2 0, E3 0, E4 0} C_DIS
LIN {X 744.142, Y -396.033, Z 108.25, A 0, B 90, C -0, E1 0, E2 0, E3 0, E4 0} C_DIS
LIN {X 743.779, Y -397.127, Z 108.25, A 0, B 90, C -0, E1 0, E2 0, E3 0, E4 0} C_DIS
LIN {X 742.809, Y -397.756, Z 108.25, A 0, B 90, C -0, E1 0, E2 0, E3 0, E4 0} C_DIS
LIN {X 737.331, Y -399.843, Z 108.25, A 0, B 90, C -0, E1 0, E2 0, E3 0, E4 0} C_DIS
LIN {X 736.468, Y -400.563, Z 108.25, A 0, B 90, C -0, E1 0, E2 0, E3 0, E4 0} C_DIS
LIN {X 736.776, Y -401.665, Z 108.25, A 0, B 90, C -0, E1 0, E2 0, E3 0, E4 0} C_DIS
LIN {X 739.55, Y -406.83, Z 108.25, A 0, B 90, C -0, E1 0, E2 0, E3 0, E4 0} C_DIS
LIN {X 739.783, Y -407.958, Z 108.25, A 0, B 90, C -0, E1 0, E2 0, E3 0, E4 0} C_DIS
LIN {X 739.257, Y -408.988, Z 108.25, A 0, B 90, C -0, E1 0, E2 0, E3 0, E4 0} C_DIS
LIN {X 735.556, Y -413.535, Z 108.25, A 0, B 90, C -0, E1 0, E2 0, E3 0, E4 0} C_DIS
LIN {X 735.169, Y -414.59, Z 108.25, A 0, B 90, C -0, E1 0, E2 0, E3 0, E4 0} C_DIS
LIN {X 735.987, Y -415.39, Z 108.25, A 0, B 90, C -0, E1 0, E2 0, E3 0, E4 0} C_DIS
LIN {X 740.971, Y -418.476, Z 108.25, A 0, B 90, C -0, E1 0, E2 0, E3 0, E4 0} C_DIS
LIN {X 741.737, Y -419.336, Z 108.25, A 0, B 90, C -0, E1 0, E2 0, E3 0, E4 0} C_DIS
LIN {X 741.797, Y -420.491, Z 108.25, A 0, B 90, C -0, E1 0, E2 0, E3 0, E4 0} C_DIS
LIN {X 740.865, Y -426.279, Z 108.25, A 0, B 90, C -0, E1 0, E2 0, E3 0, E4 0} C_DIS
LIN {X 741.058, Y -427.387, Z 108.25, A 0, B 90, C -0, E1 0, E2 0, E3 0, E4 0} C_DIS
LIN {X 742.165, Y -427.67, Z 108.25, A 0, B 90, C -0, E1 0, E2 0, E3 0, E4 0} C_DIS
LIN {X 748.025, Y -427.851, Z 108.25, A 0, B 90, C -0, E1 0, E2 0, E3 0, E4 0} C_DIS
LIN {X 749.119, Y -428.213, Z 108.25, A 0, B 90, C -0, E1 0, E2 0, E3 0, E4 0} C_DIS
LIN {X 749.748, Y -429.183, Z 108.25, A 0, B 90, C -0, E1 0, E2 0, E3 0, E4 0} C_DIS
LIN {X 751.836, Y -434.662, Z 108.25, A 0, B 90, C -0, E1 0, E2 0, E3 0, E4 0} C_DIS
LIN {X 752.556, Y -435.525, Z 108.25, A 0, B 90, C -0, E1 0, E2 0, E3 0, E4 0} C_DIS
LIN {X 753.657, Y -435.217, Z 108.25, A 0, B 90, C -0, E1 0, E2 0, E3 0, E4 0} C_DIS
LIN {X 758.822, Y -432.443, Z 108.25, A 0, B 90, C -0, E1 0, E2 0, E3 0, E4 0} C_DIS
LIN {X 759.95, Y -432.21, Z 108.25, A 0, B 90, C -0, E1 0, E2 0, E3 0, E4 0} C_DIS
LIN {X 760.98, Y -432.735, Z 108.25, A 0, B 90, C -0, E1 0, E2 0, E3 0, E4 0} C_DIS
LIN {X 765.527, Y -436.436, Z 108.25, A 0, B 90, C -0, E1 0, E2 0, E3 0, E4 0} C_DIS
LIN {X 766.583, Y -436.823, Z 108.25, A 0, B 90, C -0, E1 0, E2 0, E3 0, E4 0} C_DIS
LIN {X 767.382, Y -436.006, Z 108.25, A 0, B 90, C -0, E1 0, E2 0, E3 0, E4 0} C_DIS
LIN {X 770.468, Y -431.021, Z 108.25, A 0, B 90, C -0, E1 0, E2 0, E3 0, E4 0} C_DIS
LIN {X 771.329, Y -430.255, Z 108.25, A 0, B 90, C -0, E1 0, E2 0, E3 0, E4 0} C_DIS
LIN {X 772.484, Y -430.196, Z 108.25, A 0, B 90, C -0, E1 0, E2 0, E3 0, E4 0} C_DIS
LIN {X 778.272, Y -431.127, Z 108.25, A 0, B 90, C -0, E1 0, E2 0, E3 0, E4 0} C_DIS
LIN {X 779.379, Y -430.935, Z 108.25, A 0, B 90, C -0, E1 0, E2 0, E3 0, E4 0} C_DIS
LIN {X 779.663, Y -429.827, Z 108.25, A 0, B 90, C -0, E1 0, E2 0, E3 0, E4 0} C_DIS
LIN {X 779.843, Y -423.967, Z 108.25, A 0, B 90, C -0, E1 0, E2 0, E3 0, E4 0} C_DIS
LIN {X 780.206, Y -422.873, Z 108.25, A 0, B 90, C -0, E1 0, E2 0, E3 0, E4 0} C_DIS
LIN {X 781.176, Y -422.244, Z 108.25, A 0, B 90, C -0, E1 0, E2 0, E3 0, E4 0} C_DIS
LIN {X 786.654, Y -420.157, Z 108.25, A 0, B 90, C -0, E1 0, E2 0, E3 0, E4 0} C_DIS
LIN {X 787.517, Y -419.437, Z 108.25, A 0, B 90, C -0, E1 0, E2 0, E3 0, E4 0} C_DIS
LIN {X 787.209, Y -418.335, Z 108.25, A 0, B 90, C -0, E1 0, E2 0, E3 0, E4 0} C_DIS
LIN {X 784.435, Y -413.17, Z 108.25, A 0, B 90, C -0, E1 0, E2 0, E3 0, E4 0} C_DIS
LIN {X 784.202, Y -412.042, Z 108.25, A 0, B 90, C -0, E1 0, E2 0, E3 0, E4 0} C_DIS
LIN {X 784.728, Y -411.012, Z 108.25, A 0, B 90, C -0, E1 0, E2 0, E3 0, E4 0} C_DIS
LIN {X 788.429, Y -406.465, Z 108.25, A 0, B 90, C -0, E1 0, E2 0, E3 0, E4 0} C_DIS
LIN {X 788.816, Y -405.41, Z 108.25, A 0, B 90, C -0, E1 0, E2 0, E3 0, E4 0} C_DIS
LIN {X 787.998, Y -404.61, Z 108.25, A 0, B 90, C -0, E1 0, E2 0, E3 0, E4 0} C_DIS
LIN {X 783.014, Y -401.524, Z 108.25, A 0, B 90, C -0, E1 0, E2 0, E3 0, E4 0} C_DIS
LIN {X 782.248, Y -400.664, Z 108.25, A 0, B 90, C -0, E1 0, E2 0, E3 0, E4 0} C_DIS
LIN {X 782.188, Y -399.509, Z 108.25, A 0, B 90, C -0, E1 0, E2 0, E3 0, E4 0} C_DIS
LIN {X 783.12, Y -393.721, Z 108.25, A 0, B 90, C -0, E1 0, E2 0, E3 0, E4 0} C_DIS
LIN {X 782.927, Y -392.613, Z 108.25, A 0, B 90, C -0, E1 0, E2 0, E3 0, E4 0} C_DIS
LIN {X 781.819, Y -392.33, Z 108.25, A 0, B 90, C -0, E1 0, E2 0, E3 0, E4 0} C_DIS
LIN {X 775.959, Y -392.149, Z 108.25, A 0, B 90, C -0, E1 0, E2 0, E3 0, E4 0} C_DIS
LIN {X 774.866, Y -391.787, Z 108.25, A 0, B 90, C -0, E1 0, E2 0, E3 0, E4 0} C_DIS
LIN {X 774.237, Y -390.817, Z 108.25, A 0, B 90, C -0, E1 0, E2 0, E3 0, E4 0} C_DIS
LIN {X 772.149, Y -385.338, Z 108.25, A 0, B 90, C -0, E1 0, E2 0, E3 0, E4 0} C_DIS
LIN {X 771.429, Y -384.475, Z 108.25, A 0, B 90, C -0, E1 0, E2 0, E3 0, E4 0} C_DIS
LIN {X 770.328, Y -384.783, Z 108.25, A 0, B 90, C -0, E1 0, E2 0, E3 0, E4 0} C_DIS
LIN {X 766.196, Y -387.003, Z 108.25, A 0, B 90, C -0, E1 0, E2 0, E3 0, E4 0} C_DIS
LIN {X 764.984, Y -387.621, Z 108.9, A 0, B 90, C -0, E1 0, E2 0, E3 0, E4 0} C_DIS
LIN {X 763.862, Y -387.862, Z 108.9, A 0, B 90, C -0, E1 0, E2 0, E3 0, E4 0} C_DIS
LIN {X 762.832, Y -387.346, Z 108.9, A 0, B 90, C -0, E1 0, E2 0, E3 0, E4 0} C_DIS
LIN {X 758.275, Y -383.693, Z 108.9, A 0, B 90, C -0, E1 0, E2 0, E3 0, E4 0} C_DIS
LIN {X 757.221, Y -383.316, Z 108.9, A 0, B 90, C -0, E1 0, E2 0, E3 0, E4 0} C_DIS
LIN {X 756.431, Y -384.136, Z 108.9, A 0, B 90, C -0, E1 0, E2 0, E3 0, E4 0} C_DIS
LIN {X 753.394, Y -389.124, Z 108.9, A 0, B 90, C -0, E1 0, E2 0, E3 0, E4 0} C_DIS
LIN {X 752.542, Y -389.893, Z 108.9, A 0, B 90, C -0, E1 0, E2 0, E3 0, E4 0} C_DIS
LIN {X 751.393, Y -389.961, Z 108.9, A 0, B 90, C -0, E1 0, E2 0, E3 0, E4 0} C_DIS
LIN {X 745.62, Y -389.076, Z 108.9, A 0, B 90, C -0, E1 0, E2 0, E3 0, E4 0} C_DIS
LIN {X 744.518, Y -389.276, Z 108.9, A 0, B 90, C -0, E1 0, E2 0, E3 0, E4 0} C_DIS
LIN {X 744.244, Y -390.382, Z 108.9, A 0, B 90, C -0, E1 0, E2 0, E3 0, E4 0} C_DIS
LIN {X 744.108, Y -396.22, Z 108.9, A 0, B 90, C -0, E1 0, E2 0, E3 0, E4 0} C_DIS
LIN {X 743.755, Y -397.312, Z 108.9, A 0, B 90, C -0, E1 0, E2 0, E3 0, E4 0} C_DIS
LIN {X 742.793, Y -397.946, Z 108.9, A 0, B 90, C -0, E1 0, E2 0, E3 0, E4 0} C_DIS
LIN {X 737.352, Y -400.066, Z 108.9, A 0, B 90, C -0, E1 0, E2 0, E3 0, E4 0} C_DIS
LIN {X 736.497, Y -400.79, Z 108.9, A 0, B 90, C -0, E1 0, E2 0, E3 0, E4 0} C_DIS
LIN {X 736.813, Y -401.884, Z 108.9, A 0, B 90, C -0, E1 0, E2 0, E3 0, E4 0} C_DIS
LIN {X 739.614, Y -407.008, Z 108.9, A 0, B 90, C -0, E1 0, E2 0, E3 0, E4 0} C_DIS
LIN {X 739.854, Y -408.131, Z 108.9, A 0, B 90, C -0, E1 0, E2 0, E3 0, E4 0} C_DIS
LIN {X 739.338, Y -409.16, Z 108.9, A 0, B 90, C -0, E1 0, E2 0, E3 0, E4 0} C_DIS
LIN {X 735.686, Y -413.717, Z 108.9, A 0, B 90, C -0, E1 0, E2 0, E3 0, E4 0} C_DIS
LIN {X 735.308, Y -414.771, Z 108.9, A 0, B 90, C -0, E1 0, E2 0, E3 0, E4 0} C_DIS
LIN {X 736.128, Y -415.561, Z 108.9, A 0, B 90, C -0, E1 0, E2 0, E3 0, E4 0} C_DIS
LIN {X 741.116, Y -418.599, Z 108.9, A 0, B 90, C -0, E1 0, E2 0, E3 0, E4 0} C_DIS
LIN {X 741.886, Y -419.45, Z 108.9, A 0, B 90, C -0, E1 0, E2 0, E3 0, E4 0} C_DIS
LIN {X 741.954, Y -420.6, Z 108.9, A 0, B 90, C -0, E1 0, E2 0, E3 0, E4 0} C_DIS
LIN {X 741.069, Y -426.372, Z 108.9, A 0, B 90, C -0, E1 0, E2 0, E3 0, E4 0} C_DIS
LIN {X 741.269, Y -427.474, Z 108.9, A 0, B 90, C -0, E1 0, E2 0, E3 0, E4 0} C_DIS
LIN {X 742.374, Y -427.749, Z 108.9, A 0, B 90, C -0, E1 0, E2 0, E3 0, E4 0} C_DIS
LIN {X 748.212, Y -427.885, Z 108.9, A 0, B 90, C -0, E1 0, E2 0, E3 0, E4 0} C_DIS
LIN {X 749.305, Y -428.238, Z 108.9, A 0, B 90, C -0, E1 0, E2 0, E3 0, E4 0} C_DIS
LIN {X 749.938, Y -429.199, Z 108.9, A 0, B 90, C -0, E1 0, E2 0, E3 0, E4 0} C_DIS
LIN {X 752.058, Y -434.641, Z 108.9, A 0, B 90, C -0, E1 0, E2 0, E3 0, E4 0} C_DIS
LIN {X 752.782, Y -435.495, Z 108.9, A 0, B 90, C -0, E1 0, E2 0, E3 0, E4 0} C_DIS
LIN {X 753.877, Y -435.18, Z 108.9, A 0, B 90, C -0, E1 0, E2 0, E3 0, E4 0} C_DIS
LIN {X 759.001, Y -432.379, Z 108.9, A 0, B 90, C -0, E1 0, E2 0, E3 0, E4 0} C_DIS
LIN {X 760.123, Y -432.138, Z 108.9, A 0, B 90, C -0, E1 0, E2 0, E3 0, E4 0} C_DIS
LIN {X 761.153, Y -432.654, Z 108.9, A 0, B 90, C -0, E1 0, E2 0, E3 0, E4 0} C_DIS
LIN {X 765.71, Y -436.307, Z 108.9, A 0, B 90, C -0, E1 0, E2 0, E3 0, E4 0} C_DIS
LIN {X 766.764, Y -436.684, Z 108.9, A 0, B 90, C -0, E1 0, E2 0, E3 0, E4 0} C_DIS
LIN {X 767.554, Y -435.864, Z 108.9, A 0, B 90, C -0, E1 0, E2 0, E3 0, E4 0} C_DIS
LIN {X 770.591, Y -430.876, Z 108.9, A 0, B 90, C -0, E1 0, E2 0, E3 0, E4 0} C_DIS
LIN {X 771.443, Y -430.107, Z 108.9, A 0, B 90, C -0, E1 0, E2 0, E3 0, E4 0} C_DIS
LIN {X 772.592, Y -430.039, Z 108.9, A 0, B 90, C -0, E1 0, E2 0, E3 0, E4 0} C_DIS
LIN {X 778.365, Y -430.924, Z 108.9, A 0, B 90, C -0, E1 0, E2 0, E3 0, E4 0} C_DIS
LIN {X 779.467, Y -430.724, Z 108.9, A 0, B 90, C -0, E1 0, E2 0, E3 0, E4 0} C_DIS
LIN {X 779.741, Y -429.618, Z 108.9, A 0, B 90, C -0, E1 0, E2 0, E3 0, E4 0} C_DIS
LIN {X 779.877, Y -423.78, Z 108.9, A 0, B 90, C -0, E1 0, E2 0, E3 0, E4 0} C_DIS
LIN {X 780.23, Y -422.688, Z 108.9, A 0, B 90, C -0, E1 0, E2 0, E3 0, E4 0} C_DIS
LIN {X 781.192, Y -422.054, Z 108.9, A 0, B 90, C -0, E1 0, E2 0, E3 0, E4 0} C_DIS
LIN {X 786.633, Y -419.934, Z 108.9, A 0, B 90, C -0, E1 0, E2 0, E3 0, E4 0} C_DIS
LIN {X 787.487, Y -419.21, Z 108.9, A 0, B 90, C -0, E1 0, E2 0, E3 0, E4 0} C_DIS
LIN {X 787.172, Y -418.116, Z 108.9, A 0, B 90, C -0, E1 0, E2 0, E3 0, E4 0} C_DIS
LIN {X 784.371, Y -412.992, Z 108.9, A 0, B 90, C -0, E1 0, E2 0, E3 0, E4 0} C_DIS
LIN {X 784.131, Y -411.869, Z 108.9, A 0, B 90, C -0, E1 0, E2 0, E3 0, E4 0} C_DIS
LIN {X 784.647, Y -410.84, Z 108.9, A 0, B 90, C -0, E1 0, E2 0, E3 0, E4 0} C_DIS
LIN {X 788.299, Y -406.283, Z 108.9, A 0, B 90, C -0, E1 0, E2 0, E3 0, E4 0} C_DIS
LIN {X 788.677, Y -405.229, Z 108.9, A 0, B 90, C -0, E1 0, E2 0, E3 0, E4 0} C_DIS
LIN {X 787.857, Y -404.439, Z 108.9, A 0, B 90, C -0, E1 0, E2 0, E3 0, E4 0} C_DIS
LIN {X 782.869, Y -401.401, Z 108.9, A 0, B 90, C -0, E1 0, E2 0, E3 0, E4 0} C_DIS
LIN {X 782.099, Y -400.55, Z 108.9, A 0, B 90, C -0, E1 0, E2 0, E3 0, E4 0} C_DIS
LIN {X 782.031, Y -399.4, Z 108.9, A 0, B 90, C -0, E1 0, E2 0, E3 0, E4 0} C_DIS
LIN {X 782.916, Y -393.628, Z 108.9, A 0, B 90, C -0, E1 0, E2 0, E3 0, E4 0} C_DIS
LIN {X 782.716, Y -392.526, Z 108.9, A 0, B 90, C -0, E1 0, E2 0, E3 0, E4 0} C_DIS
LIN {X 781.611, Y -392.251, Z 108.9, A 0, B 90, C -0, E1 0, E2 0, E3 0, E4 0} C_DIS
LIN {X 775.773, Y -392.115, Z 108.9, A 0, B 90, C -0, E1 0, E2 0, E3 0, E4 0} C_DIS
LIN {X 774.68, Y -391.762, Z 108.9, A 0, B 90, C -0, E1 0, E2 0, E3 0, E4 0} C_DIS
LIN {X 774.047, Y -390.801, Z 108.9, A 0, B 90, C -0, E1 0, E2 0, E3 0, E4 0} C_DIS
LIN {X 771.927, Y -385.359, Z 108.9, A 0, B 90, C -0, E1 0, E2 0, E3 0, E4 0} C_DIS
LIN {X 771.203, Y -384.505, Z 108.9, A 0, B 90, C -0, E1 0, E2 0, E3 0, E4 0} C_DIS
LIN {X 770.108, Y -384.82, Z 108.9, A 0, B 90, C -0, E1 0, E2 0, E3 0, E4 0} C_DIS
LIN {X 766.009, Y -387.061, Z 108.9, A 0, B 90, C -0, E1 0, E2 0, E3 0, E4 0} C_DIS
LIN {X 764.808, Y -387.686, Z 109.55, A 0, B 90, C -0, E1 0, E2 0, E3 0, E4 0} C_DIS
LIN {X 763.691, Y -387.933, Z 109.55, A 0, B 90, C -0, E1 0, E2 0, E3 0, E4 0} C_DIS
LIN {X 762.662, Y -387.427, Z 109.55, A 0, B 90, C -0, E1 0, E2 0, E3 0, E4 0} C_DIS
LIN {X 758.096, Y -383.822, Z 109.55, A 0, B 90, C -0, E1 0, E2 0, E3 0, E4 0} C_DIS
LIN {X 757.043, Y -383.453, Z 109.55, A 0, B 90, C -0, E1 0, E2 0, E3 0, E4 0} C_DIS
LIN {X 756.262, Y -384.276, Z 109.55, A 0, B 90, C -0, E1 0, E2 0, E3 0, E4 0} C_DIS
LIN {X 753.273, Y -389.268, Z 109.55, A 0, B 90, C -0, E1 0, E2 0, E3 0, E4 0} C_DIS
LIN {X 752.431, Y -390.04, Z 109.55, A 0, B 90, C -0, E1 0, E2 0, E3 0, E4 0} C_DIS
LIN {X 751.286, Y -390.117, Z 109.55, A 0, B 90, C -0, E1 0, E2 0, E3 0, E4 0} C_DIS
LIN {X 745.529, Y -389.277, Z 109.55, A 0, B 90, C -0, E1 0, E2 0, E3 0, E4 0} C_DIS
LIN {X 744.433, Y -389.485, Z 109.55, A 0, B 90, C -0, E1 0, E2 0, E3 0, E4 0} C_DIS
LIN {X 744.168, Y -390.588, Z 109.55, A 0, B 90, C -0, E1 0, E2 0, E3 0, E4 0} C_DIS
LIN {X 744.075, Y -396.405, Z 109.55, A 0, B 90, C -0, E1 0, E2 0, E3 0, E4 0} C_DIS
LIN {X 743.732, Y -397.495, Z 109.55, A 0, B 90, C -0, E1 0, E2 0, E3 0, E4 0} C_DIS
LIN {X 742.778, Y -398.134, Z 109.55, A 0, B 90, C -0, E1 0, E2 0, E3 0, E4 0} C_DIS
LIN {X 737.373, Y -400.286, Z 109.55, A 0, B 90, C -0, E1 0, E2 0, E3 0, E4 0} C_DIS
LIN {X 736.528, Y -401.013, Z 109.55, A 0, B 90, C -0, E1 0, E2 0, E3 0, E4 0} C_DIS
LIN {X 736.85, Y -402.101, Z 109.55, A 0, B 90, C -0, E1 0, E2 0, E3 0, E4 0} C_DIS
LIN {X 739.678, Y -407.185, Z 109.55, A 0, B 90, C -0, E1 0, E2 0, E3 0, E4 0} C_DIS
LIN {X 739.926, Y -408.301, Z 109.55, A 0, B 90, C -0, E1 0, E2 0, E3 0, E4 0} C_DIS
LIN {X 739.419, Y -409.331, Z 109.55, A 0, B 90, C -0, E1 0, E2 0, E3 0, E4 0} C_DIS
LIN {X 735.814, Y -413.897, Z 109.55, A 0, B 90, C -0, E1 0, E2 0, E3 0, E4 0} C_DIS
LIN {X 735.446, Y -414.949, Z 109.55, A 0, B 90, C -0, E1 0, E2 0, E3 0, E4 0} C_DIS
LIN {X 736.269, Y -415.731, Z 109.55, A 0, B 90, C -0, E1 0, E2 0, E3 0, E4 0} C_DIS
LIN {X 741.26, Y -418.719, Z 109.55, A 0, B 90, C -0, E1 0, E2 0, E3 0, E4 0} C_DIS
LIN {X 742.033, Y -419.562, Z 109.55, A 0, B 90, C -0, E1 0, E2 0, E3 0, E4 0} C_DIS
LIN {X 742.109, Y -420.707, Z 109.55, A 0, B 90, C -0, E1 0, E2 0, E3 0, E4 0} C_DIS
LIN {X 741.27, Y -426.464, Z 109.55, A 0, B 90, C -0, E1 0, E2 0, E3 0, E4 0} C_DIS
LIN {X 741.477, Y -427.56, Z 109.55, A 0, B 90, C -0, E1 0, E2 0, E3 0, E4 0} C_DIS
LIN {X 742.58, Y -427.825, Z 109.55, A 0, B 90, C -0, E1 0, E2 0, E3 0, E4 0} C_DIS
LIN {X 748.397, Y -427.917, Z 109.55, A 0, B 90, C -0, E1 0, E2 0, E3 0, E4 0} C_DIS
LIN {X 749.488, Y -428.261, Z 109.55, A 0, B 90, C -0, E1 0, E2 0, E3 0, E4 0} C_DIS
LIN {X 750.126, Y -429.214, Z 109.55, A 0, B 90, C -0, E1 0, E2 0, E3 0, E4 0} C_DIS
LIN {X 752.278, Y -434.619, Z 109.55, A 0, B 90, C -0, E1 0, E2 0, E3 0, E4 0} C_DIS
LIN {X 753.005, Y -435.465, Z 109.55, A 0, B 90, C -0, E1 0, E2 0, E3 0, E4 0} C_DIS
LIN {X 754.093, Y -435.143, Z 109.55, A 0, B 90, C -0, E1 0, E2 0, E3 0, E4 0} C_DIS
LIN {X 759.177, Y -432.314, Z 109.55, A 0, B 90, C -0, E1 0, E2 0, E3 0, E4 0} C_DIS
LIN {X 760.294, Y -432.067, Z 109.55, A 0, B 90, C -0, E1 0, E2 0, E3 0, E4 0} C_DIS
LIN {X 761.323, Y -432.573, Z 109.55, A 0, B 90, C -0, E1 0, E2 0, E3 0, E4 0} C_DIS
LIN {X 765.889, Y -436.178, Z 109.55, A 0, B 90, C -0, E1 0, E2 0, E3 0, E4 0} C_DIS
LIN {X 766.942, Y -436.547, Z 109.55, A 0, B 90, C -0, E1 0, E2 0, E3 0, E4 0} C_DIS
LIN {X 767.723, Y -435.724, Z 109.55, A 0, B 90, C -0, E1 0, E2 0, E3 0, E4 0} C_DIS
LIN {X 770.712, Y -430.732, Z 109.55, A 0, B 90, C -0, E1 0, E2 0, E3 0, E4 0} C_DIS
LIN {X 771.554, Y -429.96, Z 109.55, A 0, B 90, C -0, E1 0, E2 0, E3 0, E4 0} C_DIS
LIN {X 772.699, Y -429.883, Z 109.55, A 0, B 90, C -0, E1 0, E2 0, E3 0, E4 0} C_DIS
LIN {X 778.456, Y -430.723, Z 109.55, A 0, B 90, C -0, E1 0, E2 0, E3 0, E4 0} C_DIS
LIN {X 779.552, Y -430.515, Z 109.55, A 0, B 90, C -0, E1 0, E2 0, E3 0, E4 0} C_DIS
LIN {X 779.817, Y -429.412, Z 109.55, A 0, B 90, C -0, E1 0, E2 0, E3 0, E4 0} C_DIS
LIN {X 779.91, Y -423.595, Z 109.55, A 0, B 90, C -0, E1 0, E2 0, E3 0, E4 0} C_DIS
LIN {X 780.253, Y -422.505, Z 109.55, A 0, B 90, C -0, E1 0, E2 0, E3 0, E4 0} C_DIS
LIN {X 781.206, Y -421.866, Z 109.55, A 0, B 90, C -0, E1 0, E2 0, E3 0, E4 0} C_DIS
LIN {X 786.612, Y -419.714, Z 109.55, A 0, B 90, C -0, E1 0, E2 0, E3 0, E4 0} C_DIS
LIN {X 787.457, Y -418.987, Z 109.55, A 0, B 90, C -0, E1 0, E2 0, E3 0, E4 0} C_DIS
LIN {X 787.135, Y -417.899, Z 109.55, A 0, B 90, C -0, E1 0, E2 0, E3 0, E4 0} C_DIS
LIN {X 784.307, Y -412.815, Z 109.55, A 0, B 90, C -0, E1 0, E2 0, E3 0, E4 0} C_DIS
LIN {X 784.059, Y -411.699, Z 109.55, A 0, B 90, C -0, E1 0, E2 0, E3 0, E4 0} C_DIS
LIN {X 784.565, Y -410.669, Z 109.55, A 0, B 90, C -0, E1 0, E2 0, E3 0, E4 0} C_DIS
LIN {X 788.171, Y -406.103, Z 109.55, A 0, B 90, C -0, E1 0, E2 0, E3 0, E4 0} C_DIS
LIN {X 788.539, Y -405.051, Z 109.55, A 0, B 90, C -0, E1 0, E2 0, E3 0, E4 0} C_DIS
LIN {X 787.716, Y -404.269, Z 109.55, A 0, B 90, C -0, E1 0, E2 0, E3 0, E4 0} C_DIS
LIN {X 782.725, Y -401.281, Z 109.55, A 0, B 90, C -0, E1 0, E2 0, E3 0, E4 0} C_DIS
LIN {X 781.952, Y -400.438, Z 109.55, A 0, B 90, C -0, E1 0, E2 0, E3 0, E4 0} C_DIS
LIN {X 781.876, Y -399.293, Z 109.55, A 0, B 90, C -0, E1 0, E2 0, E3 0, E4 0} C_DIS
LIN {X 782.715, Y -393.536, Z 109.55, A 0, B 90, C -0, E1 0, E2 0, E3 0, E4 0} C_DIS
LIN {X 782.508, Y -392.44, Z 109.55, A 0, B 90, C -0, E1 0, E2 0, E3 0, E4 0} C_DIS
LIN {X 781.405, Y -392.175, Z 109.55, A 0, B 90, C -0, E1 0, E2 0, E3 0, E4 0} C_DIS
LIN {X 775.588, Y -392.083, Z 109.55, A 0, B 90, C -0, E1 0, E2 0, E3 0, E4 0} C_DIS
LIN {X 774.497, Y -391.739, Z 109.55, A 0, B 90, C -0, E1 0, E2 0, E3 0, E4 0} C_DIS
LIN {X 773.859, Y -390.786, Z 109.55, A 0, B 90, C -0, E1 0, E2 0, E3 0, E4 0} C_DIS
LIN {X 771.707, Y -385.381, Z 109.55, A 0, B 90, C -0, E1 0, E2 0, E3 0, E4 0} C_DIS
LIN {X 770.979, Y -384.535, Z 109.55, A 0, B 90, C -0, E1 0, E2 0, E3 0, E4 0} C_DIS
LIN {X 769.891, Y -384.857, Z 109.55, A 0, B 90, C -0, E1 0, E2 0, E3 0, E4 0} C_DIS
LIN {X 765.824, Y -387.12, Z 109.55, A 0, B 90, C -0, E1 0, E2 0, E3 0, E4 0} C_DIS
LIN {X 764.634, Y -387.75, Z 110.2, A 0, B 90, C -0, E1 0, E2 0, E3 0, E4 0} C_DIS
LIN {X 763.523, Y -388.005, Z 110.2, A 0, B 90, C -0, E1 0, E2 0, E3 0, E4 0} C_DIS
LIN {X 762.494, Y -387.508, Z 110.2, A 0, B 90, C -0, E1 0, E2 0, E3 0, E4 0} C_DIS
LIN {X 757.919, Y -383.95, Z 110.2, A 0, B 90, C -0, E1 0, E2 0, E3 0, E4 0} C_DIS
LIN {X 756.868, Y -383.591, Z 110.2, A 0, B 90, C -0, E1 0, E2 0, E3 0, E4 0} C_DIS
LIN {X 756.095, Y -384.416, Z 110.2, A 0, B 90, C -0, E1 0, E2 0, E3 0, E4 0} C_DIS
LIN {X 753.155, Y -389.41, Z 110.2, A 0, B 90, C -0, E1 0, E2 0, E3 0, E4 0} C_DIS
LIN {X 752.321, Y -390.186, Z 110.2, A 0, B 90, C -0, E1 0, E2 0, E3 0, E4 0} C_DIS
LIN {X 751.181, Y -390.27, Z 110.2, A 0, B 90, C -0, E1 0, E2 0, E3 0, E4 0} C_DIS
LIN {X 745.44, Y -389.477, Z 110.2, A 0, B 90, C -0, E1 0, E2 0, E3 0, E4 0} C_DIS
LIN {X 744.35, Y -389.691, Z 110.2, A 0, B 90, C -0, E1 0, E2 0, E3 0, E4 0} C_DIS
LIN {X 744.093, Y -390.792, Z 110.2, A 0, B 90, C -0, E1 0, E2 0, E3 0, E4 0} C_DIS
LIN {X 744.044, Y -396.588, Z 110.2, A 0, B 90, C -0, E1 0, E2 0, E3 0, E4 0} C_DIS
LIN {X 743.71, Y -397.676, Z 110.2, A 0, B 90, C -0, E1 0, E2 0, E3 0, E4 0} C_DIS
LIN {X 742.765, Y -398.319, Z 110.2, A 0, B 90, C -0, E1 0, E2 0, E3 0, E4 0} C_DIS
LIN {X 737.396, Y -400.503, Z 110.2, A 0, B 90, C -0, E1 0, E2 0, E3 0, E4 0} C_DIS
LIN {X 736.559, Y -401.234, Z 110.2, A 0, B 90, C -0, E1 0, E2 0, E3 0, E4 0} C_DIS
LIN {X 736.888, Y -402.315, Z 110.2, A 0, B 90, C -0, E1 0, E2 0, E3 0, E4 0} C_DIS
LIN {X 739.742, Y -407.359, Z 110.2, A 0, B 90, C -0, E1 0, E2 0, E3 0, E4 0} C_DIS
LIN {X 739.997, Y -408.469, Z 110.2, A 0, B 90, C -0, E1 0, E2 0, E3 0, E4 0} C_DIS
LIN {X 739.5, Y -409.498, Z 110.2, A 0, B 90, C -0, E1 0, E2 0, E3 0, E4 0} C_DIS
LIN {X 735.942, Y -414.073, Z 110.2, A 0, B 90, C -0, E1 0, E2 0, E3 0, E4 0} C_DIS
LIN {X 735.583, Y -415.125, Z 110.2, A 0, B 90, C -0, E1 0, E2 0, E3 0, E4 0} C_DIS
LIN {X 736.408, Y -415.897, Z 110.2, A 0, B 90, C -0, E1 0, E2 0, E3 0, E4 0} C_DIS
LIN {X 741.403, Y -418.838, Z 110.2, A 0, B 90, C -0, E1 0, E2 0, E3 0, E4 0} C_DIS
LIN {X 742.179, Y -419.672, Z 110.2, A 0, B 90, C -0, E1 0, E2 0, E3 0, E4 0} C_DIS
LIN {X 742.263, Y -420.812, Z 110.2, A 0, B 90, C -0, E1 0, E2 0, E3 0, E4 0} C_DIS
LIN {X 741.469, Y -426.553, Z 110.2, A 0, B 90, C -0, E1 0, E2 0, E3 0, E4 0} C_DIS
LIN {X 741.684, Y -427.643, Z 110.2, A 0, B 90, C -0, E1 0, E2 0, E3 0, E4 0} C_DIS
LIN {X 742.785, Y -427.899, Z 110.2, A 0, B 90, C -0, E1 0, E2 0, E3 0, E4 0} C_DIS
LIN {X 748.58, Y -427.949, Z 110.2, A 0, B 90, C -0, E1 0, E2 0, E3 0, E4 0} C_DIS
LIN {X 749.669, Y -428.283, Z 110.2, A 0, B 90, C -0, E1 0, E2 0, E3 0, E4 0} C_DIS
LIN {X 750.312, Y -429.228, Z 110.2, A 0, B 90, C -0, E1 0, E2 0, E3 0, E4 0} C_DIS
LIN {X 752.495, Y -434.597, Z 110.2, A 0, B 90, C -0, E1 0, E2 0, E3 0, E4 0} C_DIS
LIN {X 753.226, Y -435.434, Z 110.2, A 0, B 90, C -0, E1 0, E2 0, E3 0, E4 0} C_DIS
LIN {X 754.307, Y -435.105, Z 110.2, A 0, B 90, C -0, E1 0, E2 0, E3 0, E4 0} C_DIS
LIN {X 759.351, Y -432.25, Z 110.2, A 0, B 90, C -0, E1 0, E2 0, E3 0, E4 0} C_DIS
LIN {X 760.461, Y -431.995, Z 110.2, A 0, B 90, C -0, E1 0, E2 0, E3 0, E4 0} C_DIS
LIN {X 761.491, Y -432.492, Z 110.2, A 0, B 90, C -0, E1 0, E2 0, E3 0, E4 0} C_DIS
LIN {X 766.066, Y -436.05, Z 110.2, A 0, B 90, C -0, E1 0, E2 0, E3 0, E4 0} C_DIS
LIN {X 767.117, Y -436.409, Z 110.2, A 0, B 90, C -0, E1 0, E2 0, E3 0, E4 0} C_DIS
LIN {X 767.89, Y -435.584, Z 110.2, A 0, B 90, C -0, E1 0, E2 0, E3 0, E4 0} C_DIS
LIN {X 770.83, Y -430.59, Z 110.2, A 0, B 90, C -0, E1 0, E2 0, E3 0, E4 0} C_DIS
LIN {X 771.664, Y -429.814, Z 110.2, A 0, B 90, C -0, E1 0, E2 0, E3 0, E4 0} C_DIS
LIN {X 772.804, Y -429.73, Z 110.2, A 0, B 90, C -0, E1 0, E2 0, E3 0, E4 0} C_DIS
LIN {X 778.545, Y -430.523, Z 110.2, A 0, B 90, C -0, E1 0, E2 0, E3 0, E4 0} C_DIS
LIN {X 779.635, Y -430.309, Z 110.2, A 0, B 90, C -0, E1 0, E2 0, E3 0, E4 0} C_DIS
LIN {X 779.891, Y -429.208, Z 110.2, A 0, B 90, C -0, E1 0, E2 0, E3 0, E4 0} C_DIS
LIN {X 779.941, Y -423.412, Z 110.2, A 0, B 90, C -0, E1 0, E2 0, E3 0, E4 0} C_DIS
LIN {X 780.275, Y -422.324, Z 110.2, A 0, B 90, C -0, E1 0, E2 0, E3 0, E4 0} C_DIS
LIN {X 781.22, Y -421.681, Z 110.2, A 0, B 90, C -0, E1 0, E2 0, E3 0, E4 0} C_DIS
LIN {X 786.589, Y -419.497, Z 110.2, A 0, B 90, C -0, E1 0, E2 0, E3 0, E4 0} C_DIS
LIN {X 787.426, Y -418.766, Z 110.2, A 0, B 90, C -0, E1 0, E2 0, E3 0, E4 0} C_DIS
LIN {X 787.097, Y -417.685, Z 110.2, A 0, B 90, C -0, E1 0, E2 0, E3 0, E4 0} C_DIS
LIN {X 784.243, Y -412.641, Z 110.2, A 0, B 90, C -0, E1 0, E2 0, E3 0, E4 0} C_DIS
LIN {X 783.988, Y -411.531, Z 110.2, A 0, B 90, C -0, E1 0, E2 0, E3 0, E4 0} C_DIS
LIN {X 784.485, Y -410.502, Z 110.2, A 0, B 90, C -0, E1 0, E2 0, E3 0, E4 0} C_DIS
LIN {X 788.043, Y -405.927, Z 110.2, A 0, B 90, C -0, E1 0, E2 0, E3 0, E4 0} C_DIS
LIN {X 788.402, Y -404.875, Z 110.2, A 0, B 90, C -0, E1 0, E2 0, E3 0, E4 0} C_DIS
LIN {X 787.577, Y -404.103, Z 110.2, A 0, B 90, C -0, E1 0, E2 0, E3 0, E4 0} C_DIS
LIN {X 782.582, Y -401.162, Z 110.2, A 0, B 90, C -0, E1 0, E2 0, E3 0, E4 0} C_DIS
LIN {X 781.806, Y -400.328, Z 110.2, A 0, B 90, C -0, E1 0, E2 0, E3 0, E4 0} C_DIS
LIN {X 781.722, Y -399.188, Z 110.2, A 0, B 90, C -0, E1 0, E2 0, E3 0, E4 0} C_DIS
LIN {X 782.516, Y -393.447, Z 110.2, A 0, B 90, C -0, E1 0, E2 0, E3 0, E4 0} C_DIS
LIN {X 782.301, Y -392.357, Z 110.2, A 0, B 90, C -0, E1 0, E2 0, E3 0, E4 0} C_DIS
LIN {X 781.2, Y -392.101, Z 110.2, A 0, B 90, C -0, E1 0, E2 0, E3 0, E4 0} C_DIS
LIN {X 775.405, Y -392.051, Z 110.2, A 0, B 90, C -0, E1 0, E2 0, E3 0, E4 0} C_DIS
LIN {X 774.316, Y -391.717, Z 110.2, A 0, B 90, C -0, E1 0, E2 0, E3 0, E4 0} C_DIS
LIN {X 773.673, Y -390.772, Z 110.2, A 0, B 90, C -0, E1 0, E2 0, E3 0, E4 0} C_DIS
LIN {X 771.49, Y -385.403, Z 110.2, A 0, B 90, C -0, E1 0, E2 0, E3 0, E4 0} C_DIS
LIN {X 770.759, Y -384.566, Z 110.2, A 0, B 90, C -0, E1 0, E2 0, E3 0, E4 0} C_DIS
LIN {X 769.677, Y -384.895, Z 110.2, A 0, B 90, C -0, E1 0, E2 0, E3 0, E4 0} C_DIS
LIN {X 765.642, Y -387.179, Z 110.2, A 0, B 90, C -0, E1 0, E2 0, E3 0, E4 0} C_DIS
LIN {X 764.462, Y -387.814, Z 110.85, A 0, B 90, C -0, E1 0, E2 0, E3 0, E4 0} C_DIS
LIN {X 763.358, Y -388.076, Z 110.85, A 0, B 90, C -0, E1 0, E2 0, E3 0, E4 0} C_DIS
LIN {X 762.329, Y -387.588, Z 110.85, A 0, B 90, C -0, E1 0, E2 0, E3 0, E4 0} C_DIS
LIN {X 757.745, Y -384.077, Z 110.85, A 0, B 90, C -0, E1 0, E2 0, E3 0, E4 0} C_DIS
LIN {X 756.695, Y -383.727, Z 110.85, A 0, B 90, C -0, E1 0, E2 0, E3 0, E4 0} C_DIS
LIN {X 755.932, Y -384.555, Z 110.85, A 0, B 90, C -0, E1 0, E2 0, E3 0, E4 0} C_DIS
LIN {X 753.038, Y -389.552, Z 110.85, A 0, B 90, C -0, E1 0, E2 0, E3 0, E4 0} C_DIS
LIN {X 752.213, Y -390.331, Z 110.85, A 0, B 90, C -0, E1 0, E2 0, E3 0, E4 0} C_DIS
LIN {X 751.078, Y -390.423, Z 110.85, A 0, B 90, C -0, E1 0, E2 0, E3 0, E4 0} C_DIS
LIN {X 745.353, Y -389.674, Z 110.85, A 0, B 90, C -0, E1 0, E2 0, E3 0, E4 0} C_DIS
LIN {X 744.268, Y -389.895, Z 110.85, A 0, B 90, C -0, E1 0, E2 0, E3 0, E4 0} C_DIS
LIN {X 744.021, Y -390.994, Z 110.85, A 0, B 90, C -0, E1 0, E2 0, E3 0, E4 0} C_DIS
LIN {X 744.014, Y -396.768, Z 110.85, A 0, B 90, C -0, E1 0, E2 0, E3 0, E4 0} C_DIS
LIN {X 743.689, Y -397.855, Z 110.85, A 0, B 90, C -0, E1 0, E2 0, E3 0, E4 0} C_DIS
LIN {X 742.752, Y -398.503, Z 110.85, A 0, B 90, C -0, E1 0, E2 0, E3 0, E4 0} C_DIS
LIN {X 737.419, Y -400.717, Z 110.85, A 0, B 90, C -0, E1 0, E2 0, E3 0, E4 0} C_DIS
LIN {X 736.59, Y -401.451, Z 110.85, A 0, B 90, C -0, E1 0, E2 0, E3 0, E4 0} C_DIS
LIN {X 736.926, Y -402.526, Z 110.85, A 0, B 90, C -0, E1 0, E2 0, E3 0, E4 0} C_DIS
LIN {X 739.806, Y -407.53, Z 110.85, A 0, B 90, C -0, E1 0, E2 0, E3 0, E4 0} C_DIS
LIN {X 740.069, Y -408.634, Z 110.85, A 0, B 90, C -0, E1 0, E2 0, E3 0, E4 0} C_DIS
LIN {X 739.581, Y -409.664, Z 110.85, A 0, B 90, C -0, E1 0, E2 0, E3 0, E4 0} C_DIS
LIN {X 736.07, Y -414.247, Z 110.85, A 0, B 90, C -0, E1 0, E2 0, E3 0, E4 0} C_DIS
LIN {X 735.719, Y -415.298, Z 110.85, A 0, B 90, C -0, E1 0, E2 0, E3 0, E4 0} C_DIS
LIN {X 736.547, Y -416.061, Z 110.85, A 0, B 90, C -0, E1 0, E2 0, E3 0, E4 0} C_DIS
LIN {X 741.544, Y -418.954, Z 110.85, A 0, B 90, C -0, E1 0, E2 0, E3 0, E4 0} C_DIS
LIN {X 742.323, Y -419.779, Z 110.85, A 0, B 90, C -0, E1 0, E2 0, E3 0, E4 0} C_DIS
LIN {X 742.415, Y -420.914, Z 110.85, A 0, B 90, C -0, E1 0, E2 0, E3 0, E4 0} C_DIS
LIN {X 741.666, Y -426.64, Z 110.85, A 0, B 90, C -0, E1 0, E2 0, E3 0, E4 0} C_DIS
LIN {X 741.888, Y -427.724, Z 110.85, A 0, B 90, C -0, E1 0, E2 0, E3 0, E4 0} C_DIS
LIN {X 742.987, Y -427.972, Z 110.85, A 0, B 90, C -0, E1 0, E2 0, E3 0, E4 0} C_DIS
LIN {X 748.761, Y -427.979, Z 110.85, A 0, B 90, C -0, E1 0, E2 0, E3 0, E4 0} C_DIS
LIN {X 749.848, Y -428.304, Z 110.85, A 0, B 90, C -0, E1 0, E2 0, E3 0, E4 0} C_DIS
LIN {X 750.495, Y -429.241, Z 110.85, A 0, B 90, C -0, E1 0, E2 0, E3 0, E4 0} C_DIS
LIN {X 752.709, Y -434.574, Z 110.85, A 0, B 90, C -0, E1 0, E2 0, E3 0, E4 0} C_DIS
LIN {X 753.444, Y -435.402, Z 110.85, A 0, B 90, C -0, E1 0, E2 0, E3 0, E4 0} C_DIS
LIN {X 754.519, Y -435.067, Z 110.85, A 0, B 90, C -0, E1 0, E2 0, E3 0, E4 0} C_DIS
LIN {X 759.523, Y -432.186, Z 110.85, A 0, B 90, C -0, E1 0, E2 0, E3 0, E4 0} C_DIS
LIN {X 760.627, Y -431.924, Z 110.85, A 0, B 90, C -0, E1 0, E2 0, E3 0, E4 0} C_DIS
LIN {X 761.656, Y -432.412, Z 110.85, A 0, B 90, C -0, E1 0, E2 0, E3 0, E4 0} C_DIS
LIN {X 766.24, Y -435.923, Z 110.85, A 0, B 90, C -0, E1 0, E2 0, E3 0, E4 0} C_DIS
LIN {X 767.29, Y -436.273, Z 110.85, A 0, B 90, C -0, E1 0, E2 0, E3 0, E4 0} C_DIS
LIN {X 768.053, Y -435.445, Z 110.85, A 0, B 90, C -0, E1 0, E2 0, E3 0, E4 0} C_DIS
LIN {X 770.947, Y -430.448, Z 110.85, A 0, B 90, C -0, E1 0, E2 0, E3 0, E4 0} C_DIS
LIN {X 771.772, Y -429.669, Z 110.85, A 0, B 90, C -0, E1 0, E2 0, E3 0, E4 0} C_DIS
LIN {X 772.907, Y -429.577, Z 110.85, A 0, B 90, C -0, E1 0, E2 0, E3 0, E4 0} C_DIS
LIN {X 778.632, Y -430.326, Z 110.85, A 0, B 90, C -0, E1 0, E2 0, E3 0, E4 0} C_DIS
LIN {X 779.717, Y -430.105, Z 110.85, A 0, B 90, C -0, E1 0, E2 0, E3 0, E4 0} C_DIS
LIN {X 779.964, Y -429.006, Z 110.85, A 0, B 90, C -0, E1 0, E2 0, E3 0, E4 0} C_DIS
LIN {X 779.971, Y -423.232, Z 110.85, A 0, B 90, C -0, E1 0, E2 0, E3 0, E4 0} C_DIS
LIN {X 780.296, Y -422.145, Z 110.85, A 0, B 90, C -0, E1 0, E2 0, E3 0, E4 0} C_DIS
LIN {X 781.233, Y -421.497, Z 110.85, A 0, B 90, C -0, E1 0, E2 0, E3 0, E4 0} C_DIS
LIN {X 786.566, Y -419.283, Z 110.85, A 0, B 90, C -0, E1 0, E2 0, E3 0, E4 0} C_DIS
LIN {X 787.395, Y -418.549, Z 110.85, A 0, B 90, C -0, E1 0, E2 0, E3 0, E4 0} C_DIS
LIN {X 787.059, Y -417.474, Z 110.85, A 0, B 90, C -0, E1 0, E2 0, E3 0, E4 0} C_DIS
LIN {X 784.179, Y -412.47, Z 110.85, A 0, B 90, C -0, E1 0, E2 0, E3 0, E4 0} C_DIS
LIN {X 783.916, Y -411.366, Z 110.85, A 0, B 90, C -0, E1 0, E2 0, E3 0, E4 0} C_DIS
LIN {X 784.404, Y -410.336, Z 110.85, A 0, B 90, C -0, E1 0, E2 0, E3 0, E4 0} C_DIS
LIN {X 787.915, Y -405.753, Z 110.85, A 0, B 90, C -0, E1 0, E2 0, E3 0, E4 0} C_DIS
LIN {X 788.266, Y -404.702, Z 110.85, A 0, B 90, C -0, E1 0, E2 0, E3 0, E4 0} C_DIS
LIN {X 787.438, Y -403.939, Z 110.85, A 0, B 90, C -0, E1 0, E2 0, E3 0, E4 0} C_DIS
LIN {X 782.441, Y -401.046, Z 110.85, A 0, B 90, C -0, E1 0, E2 0, E3 0, E4 0} C_DIS
LIN {X 781.662, Y -400.221, Z 110.85, A 0, B 90, C -0, E1 0, E2 0, E3 0, E4 0} C_DIS
LIN {X 781.57, Y -399.086, Z 110.85, A 0, B 90, C -0, E1 0, E2 0, E3 0, E4 0} C_DIS
LIN {X 782.319, Y -393.36, Z 110.85, A 0, B 90, C -0, E1 0, E2 0, E3 0, E4 0} C_DIS
LIN {X 782.097, Y -392.276, Z 110.85, A 0, B 90, C -0, E1 0, E2 0, E3 0, E4 0} C_DIS
LIN {X 780.998, Y -392.028, Z 110.85, A 0, B 90, C -0, E1 0, E2 0, E3 0, E4 0} C_DIS
LIN {X 775.224, Y -392.021, Z 110.85, A 0, B 90, C -0, E1 0, E2 0, E3 0, E4 0} C_DIS
LIN {X 774.137, Y -391.696, Z 110.85, A 0, B 90, C -0, E1 0, E2 0, E3 0, E4 0} C_DIS
LIN {X 773.49, Y -390.759, Z 110.85, A 0, B 90, C -0, E1 0, E2 0, E3 0, E4 0} C_DIS
LIN {X 771.276, Y -385.426, Z 110.85, A 0, B 90, C -0, E1 0, E2 0, E3 0, E4 0} C_DIS
LIN {X 770.541, Y -384.598, Z 110.85, A 0, B 90, C -0, E1 0, E2 0, E3 0, E4 0} C_DIS
LIN {X 769.466, Y -384.933, Z 110.85, A 0, B 90, C -0, E1 0, E2 0, E3 0, E4 0} C_DIS
LIN {X 765.463, Y -387.238, Z 110.85, A 0, B 90, C -0, E1 0, E2 0, E3 0, E4 0} C_DIS
LIN {X 764.293, Y -387.878, Z 111.5, A 0, B 90, C -0, E1 0, E2 0, E3 0, E4 0} C_DIS
LIN {X 763.195, Y -388.147, Z 111.5, A 0, B 90, C -0, E1 0, E2 0, E3 0, E4 0} C_DIS
LIN {X 762.166, Y -387.669, Z 111.5, A 0, B 90, C -0, E1 0, E2 0, E3 0, E4 0} C_DIS
LIN {X 757.574, Y -384.203, Z 111.5, A 0, B 90, C -0, E1 0, E2 0, E3 0, E4 0} C_DIS
LIN {X 756.525, Y -383.862, Z 111.5, A 0, B 90, C -0, E1 0, E2 0, E3 0, E4 0} C_DIS
LIN {X 755.77, Y -384.692, Z 111.5, A 0, B 90, C -0, E1 0, E2 0, E3 0, E4 0} C_DIS
LIN {X 752.924, Y -389.692, Z 111.5, A 0, B 90, C -0, E1 0, E2 0, E3 0, E4 0} C_DIS
LIN {X 752.107, Y -390.474, Z 111.5, A 0, B 90, C -0, E1 0, E2 0, E3 0, E4 0} C_DIS
LIN {X 750.977, Y -390.574, Z 111.5, A 0, B 90, C -0, E1 0, E2 0, E3 0, E4 0} C_DIS
LIN {X 745.268, Y -389.869, Z 111.5, A 0, B 90, C -0, E1 0, E2 0, E3 0, E4 0} C_DIS
LIN {X 744.188, Y -390.097, Z 111.5, A 0, B 90, C -0, E1 0, E2 0, E3 0, E4 0} C_DIS
LIN {X 743.95, Y -391.194, Z 111.5, A 0, B 90, C -0, E1 0, E2 0, E3 0, E4 0} C_DIS
LIN {X 743.984, Y -396.947, Z 111.5, A 0, B 90, C -0, E1 0, E2 0, E3 0, E4 0} C_DIS
LIN {X 743.669, Y -398.032, Z 111.5, A 0, B 90, C -0, E1 0, E2 0, E3 0, E4 0} C_DIS
LIN {X 742.74, Y -398.684, Z 111.5, A 0, B 90, C -0, E1 0, E2 0, E3 0, E4 0} C_DIS
LIN {X 737.443, Y -400.928, Z 111.5, A 0, B 90, C -0, E1 0, E2 0, E3 0, E4 0} C_DIS
LIN {X 736.622, Y -401.666, Z 111.5, A 0, B 90, C -0, E1 0, E2 0, E3 0, E4 0} C_DIS
LIN {X 736.964, Y -402.735, Z 111.5, A 0, B 90, C -0, E1 0, E2 0, E3 0, E4 0} C_DIS
LIN {X 739.87, Y -407.7, Z 111.5, A 0, B 90, C -0, E1 0, E2 0, E3 0, E4 0} C_DIS
LIN {X 740.14, Y -408.798, Z 111.5, A 0, B 90, C -0, E1 0, E2 0, E3 0, E4 0} C_DIS
LIN {X 739.661, Y -409.826, Z 111.5, A 0, B 90, C -0, E1 0, E2 0, E3 0, E4 0} C_DIS
LIN {X 736.196, Y -414.419, Z 111.5, A 0, B 90, C -0, E1 0, E2 0, E3 0, E4 0} C_DIS
LIN {X 735.854, Y -415.467, Z 111.5, A 0, B 90, C -0, E1 0, E2 0, E3 0, E4 0} C_DIS
LIN {X 736.685, Y -416.222, Z 111.5, A 0, B 90, C -0, E1 0, E2 0, E3 0, E4 0} C_DIS
LIN {X 741.684, Y -419.069, Z 111.5, A 0, B 90, C -0, E1 0, E2 0, E3 0, E4 0} C_DIS
LIN {X 742.466, Y -419.885, Z 111.5, A 0, B 90, C -0, E1 0, E2 0, E3 0, E4 0} C_DIS
LIN {X 742.566, Y -421.015, Z 111.5, A 0, B 90, C -0, E1 0, E2 0, E3 0, E4 0} C_DIS
LIN {X 741.861, Y -426.725, Z 111.5, A 0, B 90, C -0, E1 0, E2 0, E3 0, E4 0} C_DIS
LIN {X 742.09, Y -427.804, Z 111.5, A 0, B 90, C -0, E1 0, E2 0, E3 0, E4 0} C_DIS
LIN {X 743.186, Y -428.042, Z 111.5, A 0, B 90, C -0, E1 0, E2 0, E3 0, E4 0} C_DIS
LIN {X 748.939, Y -428.008, Z 111.5, A 0, B 90, C -0, E1 0, E2 0, E3 0, E4 0} C_DIS
LIN {X 750.025, Y -428.324, Z 111.5, A 0, B 90, C -0, E1 0, E2 0, E3 0, E4 0} C_DIS
LIN {X 750.677, Y -429.253, Z 111.5, A 0, B 90, C -0, E1 0, E2 0, E3 0, E4 0} C_DIS
LIN {X 752.921, Y -434.55, Z 111.5, A 0, B 90, C -0, E1 0, E2 0, E3 0, E4 0} C_DIS
LIN {X 753.658, Y -435.37, Z 111.5, A 0, B 90, C -0, E1 0, E2 0, E3 0, E4 0} C_DIS
LIN {X 754.727, Y -435.028, Z 111.5, A 0, B 90, C -0, E1 0, E2 0, E3 0, E4 0} C_DIS
LIN {X 759.692, Y -432.122, Z 111.5, A 0, B 90, C -0, E1 0, E2 0, E3 0, E4 0} C_DIS
LIN {X 760.79, Y -431.853, Z 111.5, A 0, B 90, C -0, E1 0, E2 0, E3 0, E4 0} C_DIS
LIN {X 761.819, Y -432.331, Z 111.5, A 0, B 90, C -0, E1 0, E2 0, E3 0, E4 0} C_DIS
LIN {X 766.411, Y -435.797, Z 111.5, A 0, B 90, C -0, E1 0, E2 0, E3 0, E4 0} C_DIS
LIN {X 767.46, Y -436.138, Z 111.5, A 0, B 90, C -0, E1 0, E2 0, E3 0, E4 0} C_DIS
LIN {X 768.214, Y -435.308, Z 111.5, A 0, B 90, C -0, E1 0, E2 0, E3 0, E4 0} C_DIS
LIN {X 771.061, Y -430.308, Z 111.5, A 0, B 90, C -0, E1 0, E2 0, E3 0, E4 0} C_DIS
LIN {X 771.878, Y -429.526, Z 111.5, A 0, B 90, C -0, E1 0, E2 0, E3 0, E4 0} C_DIS
LIN {X 773.008, Y -429.426, Z 111.5, A 0, B 90, C -0, E1 0, E2 0, E3 0, E4 0} C_DIS
LIN {X 778.717, Y -430.131, Z 111.5, A 0, B 90, C -0, E1 0, E2 0, E3 0, E4 0} C_DIS
LIN {X 779.797, Y -429.903, Z 111.5, A 0, B 90, C -0, E1 0, E2 0, E3 0, E4 0} C_DIS
LIN {X 780.035, Y -428.806, Z 111.5, A 0, B 90, C -0, E1 0, E2 0, E3 0, E4 0} C_DIS
LIN {X 780, Y -423.053, Z 111.5, A 0, B 90, C -0, E1 0, E2 0, E3 0, E4 0} C_DIS
LIN {X 780.316, Y -421.968, Z 111.5, A 0, B 90, C -0, E1 0, E2 0, E3 0, E4 0} C_DIS
LIN {X 781.245, Y -421.316, Z 111.5, A 0, B 90, C -0, E1 0, E2 0, E3 0, E4 0} C_DIS
LIN {X 786.542, Y -419.072, Z 111.5, A 0, B 90, C -0, E1 0, E2 0, E3 0, E4 0} C_DIS
LIN {X 787.362, Y -418.334, Z 111.5, A 0, B 90, C -0, E1 0, E2 0, E3 0, E4 0} C_DIS
LIN {X 787.021, Y -417.265, Z 111.5, A 0, B 90, C -0, E1 0, E2 0, E3 0, E4 0} C_DIS
LIN {X 784.115, Y -412.3, Z 111.5, A 0, B 90, C -0, E1 0, E2 0, E3 0, E4 0} C_DIS
LIN {X 783.845, Y -411.202, Z 111.5, A 0, B 90, C -0, E1 0, E2 0, E3 0, E4 0} C_DIS
LIN {X 784.324, Y -410.174, Z 111.5, A 0, B 90, C -0, E1 0, E2 0, E3 0, E4 0} C_DIS
LIN {X 787.789, Y -405.581, Z 111.5, A 0, B 90, C -0, E1 0, E2 0, E3 0, E4 0} C_DIS
LIN {X 788.131, Y -404.533, Z 111.5, A 0, B 90, C -0, E1 0, E2 0, E3 0, E4 0} C_DIS
LIN {X 787.3, Y -403.778, Z 111.5, A 0, B 90, C -0, E1 0, E2 0, E3 0, E4 0} C_DIS
LIN {X 782.301, Y -400.931, Z 111.5, A 0, B 90, C -0, E1 0, E2 0, E3 0, E4 0} C_DIS
LIN {X 781.519, Y -400.115, Z 111.5, A 0, B 90, C -0, E1 0, E2 0, E3 0, E4 0} C_DIS
LIN {X 781.419, Y -398.985, Z 111.5, A 0, B 90, C -0, E1 0, E2 0, E3 0, E4 0} C_DIS
LIN {X 782.124, Y -393.275, Z 111.5, A 0, B 90, C -0, E1 0, E2 0, E3 0, E4 0} C_DIS
LIN {X 781.895, Y -392.196, Z 111.5, A 0, B 90, C -0, E1 0, E2 0, E3 0, E4 0} C_DIS
LIN {X 780.799, Y -391.958, Z 111.5, A 0, B 90, C -0, E1 0, E2 0, E3 0, E4 0} C_DIS
LIN {X 775.046, Y -391.992, Z 111.5, A 0, B 90, C -0, E1 0, E2 0, E3 0, E4 0} C_DIS
LIN {X 773.96, Y -391.676, Z 111.5, A 0, B 90, C -0, E1 0, E2 0, E3 0, E4 0} C_DIS
LIN {X 773.308, Y -390.747, Z 111.5, A 0, B 90, C -0, E1 0, E2 0, E3 0, E4 0} C_DIS
LIN {X 771.064, Y -385.45, Z 111.5, A 0, B 90, C -0, E1 0, E2 0, E3 0, E4 0} C_DIS
LIN {X 770.327, Y -384.63, Z 111.5, A 0, B 90, C -0, E1 0, E2 0, E3 0, E4 0} C_DIS
LIN {X 769.258, Y -384.972, Z 111.5, A 0, B 90, C -0, E1 0, E2 0, E3 0, E4 0} C_DIS
LIN {X 765.286, Y -387.297, Z 111.5, A 0, B 90, C -0, E1 0, E2 0, E3 0, E4 0} C_DIS
LIN {X 764.126, Y -387.942, Z 112.15, A 0, B 90, C -0, E1 0, E2 0, E3 0, E4 0} C_DIS
LIN {X 763.034, Y -388.218, Z 112.15, A 0, B 90, C -0, E1 0, E2 0, E3 0, E4 0} C_DIS
LIN {X 762.006, Y -387.749, Z 112.15, A 0, B 90, C -0, E1 0, E2 0, E3 0, E4 0} C_DIS
LIN {X 757.405, Y -384.329, Z 112.15, A 0, B 90, C -0, E1 0, E2 0, E3 0, E4 0} C_DIS
LIN {X 756.358, Y -383.996, Z 112.15, A 0, B 90, C -0, E1 0, E2 0, E3 0, E4 0} C_DIS
LIN {X 755.612, Y -384.829, Z 112.15, A 0, B 90, C -0, E1 0, E2 0, E3 0, E4 0} C_DIS
LIN {X 752.811, Y -389.83, Z 112.15, A 0, B 90, C -0, E1 0, E2 0, E3 0, E4 0} C_DIS
LIN {X 752.003, Y -390.615, Z 112.15, A 0, B 90, C -0, E1 0, E2 0, E3 0, E4 0} C_DIS
LIN {X 750.878, Y -390.723, Z 112.15, A 0, B 90, C -0, E1 0, E2 0, E3 0, E4 0} C_DIS
LIN {X 745.184, Y -390.062, Z 112.15, A 0, B 90, C -0, E1 0, E2 0, E3 0, E4 0} C_DIS
LIN {X 744.111, Y -390.297, Z 112.15, A 0, B 90, C -0, E1 0, E2 0, E3 0, E4 0} C_DIS
LIN {X 743.881, Y -391.391, Z 112.15, A 0, B 90, C -0, E1 0, E2 0, E3 0, E4 0} C_DIS
LIN {X 743.956, Y -397.123, Z 112.15, A 0, B 90, C -0, E1 0, E2 0, E3 0, E4 0} C_DIS
LIN {X 743.649, Y -398.207, Z 112.15, A 0, B 90, C -0, E1 0, E2 0, E3 0, E4 0} C_DIS
LIN {X 742.729, Y -398.863, Z 112.15, A 0, B 90, C -0, E1 0, E2 0, E3 0, E4 0} C_DIS
LIN {X 737.467, Y -401.137, Z 112.15, A 0, B 90, C -0, E1 0, E2 0, E3 0, E4 0} C_DIS
LIN {X 736.655, Y -401.878, Z 112.15, A 0, B 90, C -0, E1 0, E2 0, E3 0, E4 0} C_DIS
LIN {X 737.003, Y -402.94, Z 112.15, A 0, B 90, C -0, E1 0, E2 0, E3 0, E4 0} C_DIS
LIN {X 739.934, Y -407.866, Z 112.15, A 0, B 90, C -0, E1 0, E2 0, E3 0, E4 0} C_DIS
LIN {X 740.21, Y -408.958, Z 112.15, A 0, B 90, C -0, E1 0, E2 0, E3 0, E4 0} C_DIS
LIN {X 739.741, Y -409.987, Z 112.15, A 0, B 90, C -0, E1 0, E2 0, E3 0, E4 0} C_DIS
LIN {X 736.321, Y -414.587, Z 112.15, A 0, B 90, C -0, E1 0, E2 0, E3 0, E4 0} C_DIS
LIN {X 735.989, Y -415.635, Z 112.15, A 0, B 90, C -0, E1 0, E2 0, E3 0, E4 0} C_DIS
LIN {X 736.821, Y -416.381, Z 112.15, A 0, B 90, C -0, E1 0, E2 0, E3 0, E4 0} C_DIS
LIN {X 741.823, Y -419.181, Z 112.15, A 0, B 90, C -0, E1 0, E2 0, E3 0, E4 0} C_DIS
LIN {X 742.608, Y -419.989, Z 112.15, A 0, B 90, C -0, E1 0, E2 0, E3 0, E4 0} C_DIS
LIN {X 742.716, Y -421.114, Z 112.15, A 0, B 90, C -0, E1 0, E2 0, E3 0, E4 0} C_DIS
LIN {X 742.054, Y -426.808, Z 112.15, A 0, B 90, C -0, E1 0, E2 0, E3 0, E4 0} C_DIS
LIN {X 742.29, Y -427.882, Z 112.15, A 0, B 90, C -0, E1 0, E2 0, E3 0, E4 0} C_DIS
LIN {X 743.384, Y -428.111, Z 112.15, A 0, B 90, C -0, E1 0, E2 0, E3 0, E4 0} C_DIS
LIN {X 749.116, Y -428.036, Z 112.15, A 0, B 90, C -0, E1 0, E2 0, E3 0, E4 0} C_DIS
LIN {X 750.199, Y -428.343, Z 112.15, A 0, B 90, C -0, E1 0, E2 0, E3 0, E4 0} C_DIS
LIN {X 750.856, Y -429.264, Z 112.15, A 0, B 90, C -0, E1 0, E2 0, E3 0, E4 0} C_DIS
LIN {X 753.13, Y -434.526, Z 112.15, A 0, B 90, C -0, E1 0, E2 0, E3 0, E4 0} C_DIS
LIN {X 753.87, Y -435.337, Z 112.15, A 0, B 90, C -0, E1 0, E2 0, E3 0, E4 0} C_DIS
LIN {X 754.933, Y -434.989, Z 112.15, A 0, B 90, C -0, E1 0, E2 0, E3 0, E4 0} C_DIS
LIN {X 759.859, Y -432.058, Z 112.15, A 0, B 90, C -0, E1 0, E2 0, E3 0, E4 0} C_DIS
LIN {X 760.951, Y -431.782, Z 112.15, A 0, B 90, C -0, E1 0, E2 0, E3 0, E4 0} C_DIS
LIN {X 761.979, Y -432.251, Z 112.15, A 0, B 90, C -0, E1 0, E2 0, E3 0, E4 0} C_DIS
LIN {X 766.58, Y -435.671, Z 112.15, A 0, B 90, C -0, E1 0, E2 0, E3 0, E4 0} C_DIS
LIN {X 767.627, Y -436.004, Z 112.15, A 0, B 90, C -0, E1 0, E2 0, E3 0, E4 0} C_DIS
LIN {X 768.373, Y -435.171, Z 112.15, A 0, B 90, C -0, E1 0, E2 0, E3 0, E4 0} C_DIS
LIN {X 771.174, Y -430.17, Z 112.15, A 0, B 90, C -0, E1 0, E2 0, E3 0, E4 0} C_DIS
LIN {X 771.982, Y -429.385, Z 112.15, A 0, B 90, C -0, E1 0, E2 0, E3 0, E4 0} C_DIS
LIN {X 773.107, Y -429.277, Z 112.15, A 0, B 90, C -0, E1 0, E2 0, E3 0, E4 0} C_DIS
LIN {X 778.801, Y -429.938, Z 112.15, A 0, B 90, C -0, E1 0, E2 0, E3 0, E4 0} C_DIS
LIN {X 779.874, Y -429.703, Z 112.15, A 0, B 90, C -0, E1 0, E2 0, E3 0, E4 0} C_DIS
LIN {X 780.104, Y -428.609, Z 112.15, A 0, B 90, C -0, E1 0, E2 0, E3 0, E4 0} C_DIS
LIN {X 780.028, Y -422.877, Z 112.15, A 0, B 90, C -0, E1 0, E2 0, E3 0, E4 0} C_DIS
LIN {X 780.336, Y -421.793, Z 112.15, A 0, B 90, C -0, E1 0, E2 0, E3 0, E4 0} C_DIS
LIN {X 781.256, Y -421.137, Z 112.15, A 0, B 90, C -0, E1 0, E2 0, E3 0, E4 0} C_DIS
LIN {X 786.518, Y -418.863, Z 112.15, A 0, B 90, C -0, E1 0, E2 0, E3 0, E4 0} C_DIS
LIN {X 787.33, Y -418.122, Z 112.15, A 0, B 90, C -0, E1 0, E2 0, E3 0, E4 0} C_DIS
LIN {X 786.982, Y -417.06, Z 112.15, A 0, B 90, C -0, E1 0, E2 0, E3 0, E4 0} C_DIS
LIN {X 784.051, Y -412.134, Z 112.15, A 0, B 90, C -0, E1 0, E2 0, E3 0, E4 0} C_DIS
LIN {X 783.775, Y -411.042, Z 112.15, A 0, B 90, C -0, E1 0, E2 0, E3 0, E4 0} C_DIS
LIN {X 784.244, Y -410.013, Z 112.15, A 0, B 90, C -0, E1 0, E2 0, E3 0, E4 0} C_DIS
LIN {X 787.664, Y -405.413, Z 112.15, A 0, B 90, C -0, E1 0, E2 0, E3 0, E4 0} C_DIS
LIN {X 787.996, Y -404.365, Z 112.15, A 0, B 90, C -0, E1 0, E2 0, E3 0, E4 0} C_DIS
LIN {X 787.164, Y -403.619, Z 112.15, A 0, B 90, C -0, E1 0, E2 0, E3 0, E4 0} C_DIS
LIN {X 782.162, Y -400.819, Z 112.15, A 0, B 90, C -0, E1 0, E2 0, E3 0, E4 0} C_DIS
LIN {X 781.377, Y -400.011, Z 112.15, A 0, B 90, C -0, E1 0, E2 0, E3 0, E4 0} C_DIS
LIN {X 781.269, Y -398.886, Z 112.15, A 0, B 90, C -0, E1 0, E2 0, E3 0, E4 0} C_DIS
LIN {X 781.931, Y -393.192, Z 112.15, A 0, B 90, C -0, E1 0, E2 0, E3 0, E4 0} C_DIS
LIN {X 781.695, Y -392.118, Z 112.15, A 0, B 90, C -0, E1 0, E2 0, E3 0, E4 0} C_DIS
LIN {X 780.601, Y -391.889, Z 112.15, A 0, B 90, C -0, E1 0, E2 0, E3 0, E4 0} C_DIS
LIN {X 774.869, Y -391.964, Z 112.15, A 0, B 90, C -0, E1 0, E2 0, E3 0, E4 0} C_DIS
LIN {X 773.785, Y -391.657, Z 112.15, A 0, B 90, C -0, E1 0, E2 0, E3 0, E4 0} C_DIS
LIN {X 773.129, Y -390.736, Z 112.15, A 0, B 90, C -0, E1 0, E2 0, E3 0, E4 0} C_DIS
LIN {X 770.855, Y -385.474, Z 112.15, A 0, B 90, C -0, E1 0, E2 0, E3 0, E4 0} C_DIS
LIN {X 770.115, Y -384.663, Z 112.15, A 0, B 90, C -0, E1 0, E2 0, E3 0, E4 0} C_DIS
LIN {X 769.052, Y -385.011, Z 112.15, A 0, B 90, C -0, E1 0, E2 0, E3 0, E4 0} C_DIS
LIN {X 765.111, Y -387.356, Z 112.15, A 0, B 90, C -0, E1 0, E2 0, E3 0, E4 0} C_DIS
LIN {X 763.962, Y -388.006, Z 112.8, A 0, B 90, C -0, E1 0, E2 0, E3 0, E4 0} C_DIS
LIN {X 762.876, Y -388.289, Z 112.8, A 0, B 90, C -0, E1 0, E2 0, E3 0, E4 0} C_DIS
LIN {X 761.847, Y -387.828, Z 112.8, A 0, B 90, C -0, E1 0, E2 0, E3 0, E4 0} C_DIS
LIN {X 757.239, Y -384.453, Z 112.8, A 0, B 90, C -0, E1 0, E2 0, E3 0, E4 0} C_DIS
LIN {X 756.193, Y -384.129, Z 112.8, A 0, B 90, C -0, E1 0, E2 0, E3 0, E4 0} C_DIS
LIN {X 755.456, Y -384.964, Z 112.8, A 0, B 90, C -0, E1 0, E2 0, E3 0, E4 0} C_DIS
LIN {X 752.701, Y -389.968, Z 112.8, A 0, B 90, C -0, E1 0, E2 0, E3 0, E4 0} C_DIS
LIN {X 751.901, Y -390.756, Z 112.8, A 0, B 90, C -0, E1 0, E2 0, E3 0, E4 0} C_DIS
LIN {X 750.781, Y -390.871, Z 112.8, A 0, B 90, C -0, E1 0, E2 0, E3 0, E4 0} C_DIS
LIN {X 745.103, Y -390.253, Z 112.8, A 0, B 90, C -0, E1 0, E2 0, E3 0, E4 0} C_DIS
LIN {X 744.035, Y -390.495, Z 112.8, A 0, B 90, C -0, E1 0, E2 0, E3 0, E4 0} C_DIS
LIN {X 743.814, Y -391.587, Z 112.8, A 0, B 90, C -0, E1 0, E2 0, E3 0, E4 0} C_DIS
LIN {X 743.93, Y -397.297, Z 112.8, A 0, B 90, C -0, E1 0, E2 0, E3 0, E4 0} C_DIS
LIN {X 743.631, Y -398.38, Z 112.8, A 0, B 90, C -0, E1 0, E2 0, E3 0, E4 0} C_DIS
LIN {X 742.719, Y -399.04, Z 112.8, A 0, B 90, C -0, E1 0, E2 0, E3 0, E4 0} C_DIS
LIN {X 737.492, Y -401.343, Z 112.8, A 0, B 90, C -0, E1 0, E2 0, E3 0, E4 0} C_DIS
LIN {X 736.688, Y -402.087, Z 112.8, A 0, B 90, C -0, E1 0, E2 0, E3 0, E4 0} C_DIS
LIN {X 737.043, Y -403.143, Z 112.8, A 0, B 90, C -0, E1 0, E2 0, E3 0, E4 0} C_DIS
LIN {X 739.998, Y -408.031, Z 112.8, A 0, B 90, C -0, E1 0, E2 0, E3 0, E4 0} C_DIS
LIN {X 740.281, Y -409.117, Z 112.8, A 0, B 90, C -0, E1 0, E2 0, E3 0, E4 0} C_DIS
LIN {X 739.821, Y -410.145, Z 112.8, A 0, B 90, C -0, E1 0, E2 0, E3 0, E4 0} C_DIS
LIN {X 736.446, Y -414.753, Z 112.8, A 0, B 90, C -0, E1 0, E2 0, E3 0, E4 0} C_DIS
LIN {X 736.122, Y -415.799, Z 112.8, A 0, B 90, C -0, E1 0, E2 0, E3 0, E4 0} C_DIS
LIN {X 736.957, Y -416.536, Z 112.8, A 0, B 90, C -0, E1 0, E2 0, E3 0, E4 0} C_DIS
LIN {X 741.96, Y -419.292, Z 112.8, A 0, B 90, C -0, E1 0, E2 0, E3 0, E4 0} C_DIS
LIN {X 742.748, Y -420.091, Z 112.8, A 0, B 90, C -0, E1 0, E2 0, E3 0, E4 0} C_DIS
LIN {X 742.864, Y -421.211, Z 112.8, A 0, B 90, C -0, E1 0, E2 0, E3 0, E4 0} C_DIS
LIN {X 742.245, Y -426.89, Z 112.8, A 0, B 90, C -0, E1 0, E2 0, E3 0, E4 0} C_DIS
LIN {X 742.487, Y -427.958, Z 112.8, A 0, B 90, C -0, E1 0, E2 0, E3 0, E4 0} C_DIS
LIN {X 743.579, Y -428.179, Z 112.8, A 0, B 90, C -0, E1 0, E2 0, E3 0, E4 0} C_DIS
LIN {X 749.29, Y -428.063, Z 112.8, A 0, B 90, C -0, E1 0, E2 0, E3 0, E4 0} C_DIS
LIN {X 750.372, Y -428.361, Z 112.8, A 0, B 90, C -0, E1 0, E2 0, E3 0, E4 0} C_DIS
LIN {X 751.032, Y -429.274, Z 112.8, A 0, B 90, C -0, E1 0, E2 0, E3 0, E4 0} C_DIS
LIN {X 753.336, Y -434.501, Z 112.8, A 0, B 90, C -0, E1 0, E2 0, E3 0, E4 0} C_DIS
LIN {X 754.079, Y -435.304, Z 112.8, A 0, B 90, C -0, E1 0, E2 0, E3 0, E4 0} C_DIS
LIN {X 755.135, Y -434.95, Z 112.8, A 0, B 90, C -0, E1 0, E2 0, E3 0, E4 0} C_DIS
LIN {X 760.023, Y -431.994, Z 112.8, A 0, B 90, C -0, E1 0, E2 0, E3 0, E4 0} C_DIS
LIN {X 761.109, Y -431.711, Z 112.8, A 0, B 90, C -0, E1 0, E2 0, E3 0, E4 0} C_DIS
LIN {X 762.138, Y -432.172, Z 112.8, A 0, B 90, C -0, E1 0, E2 0, E3 0, E4 0} C_DIS
LIN {X 766.746, Y -435.547, Z 112.8, A 0, B 90, C -0, E1 0, E2 0, E3 0, E4 0} C_DIS
LIN {X 767.792, Y -435.871, Z 112.8, A 0, B 90, C -0, E1 0, E2 0, E3 0, E4 0} C_DIS
LIN {X 768.529, Y -435.036, Z 112.8, A 0, B 90, C -0, E1 0, E2 0, E3 0, E4 0} C_DIS
LIN {X 771.284, Y -430.032, Z 112.8, A 0, B 90, C -0, E1 0, E2 0, E3 0, E4 0} C_DIS
LIN {X 772.083, Y -429.244, Z 112.8, A 0, B 90, C -0, E1 0, E2 0, E3 0, E4 0} C_DIS
LIN {X 773.204, Y -429.129, Z 112.8, A 0, B 90, C -0, E1 0, E2 0, E3 0, E4 0} C_DIS
LIN {X 778.882, Y -429.747, Z 112.8, A 0, B 90, C -0, E1 0, E2 0, E3 0, E4 0} C_DIS
LIN {X 779.95, Y -429.505, Z 112.8, A 0, B 90, C -0, E1 0, E2 0, E3 0, E4 0} C_DIS
LIN {X 780.171, Y -428.413, Z 112.8, A 0, B 90, C -0, E1 0, E2 0, E3 0, E4 0} C_DIS
LIN {X 780.055, Y -422.703, Z 112.8, A 0, B 90, C -0, E1 0, E2 0, E3 0, E4 0} C_DIS
LIN {X 780.354, Y -421.62, Z 112.8, A 0, B 90, C -0, E1 0, E2 0, E3 0, E4 0} C_DIS
LIN {X 781.266, Y -420.96, Z 112.8, A 0, B 90, C -0, E1 0, E2 0, E3 0, E4 0} C_DIS
LIN {X 786.493, Y -418.657, Z 112.8, A 0, B 90, C -0, E1 0, E2 0, E3 0, E4 0} C_DIS
LIN {X 787.297, Y -417.913, Z 112.8, A 0, B 90, C -0, E1 0, E2 0, E3 0, E4 0} C_DIS
LIN {X 786.942, Y -416.857, Z 112.8, A 0, B 90, C -0, E1 0, E2 0, E3 0, E4 0} C_DIS
LIN {X 783.987, Y -411.969, Z 112.8, A 0, B 90, C -0, E1 0, E2 0, E3 0, E4 0} C_DIS
LIN {X 783.704, Y -410.883, Z 112.8, A 0, B 90, C -0, E1 0, E2 0, E3 0, E4 0} C_DIS
LIN {X 784.164, Y -409.855, Z 112.8, A 0, B 90, C -0, E1 0, E2 0, E3 0, E4 0} C_DIS
LIN {X 787.539, Y -405.247, Z 112.8, A 0, B 90, C -0, E1 0, E2 0, E3 0, E4 0} C_DIS
LIN {X 787.863, Y -404.201, Z 112.8, A 0, B 90, C -0, E1 0, E2 0, E3 0, E4 0} C_DIS
LIN {X 787.028, Y -403.464, Z 112.8, A 0, B 90, C -0, E1 0, E2 0, E3 0, E4 0} C_DIS
LIN {X 782.025, Y -400.708, Z 112.8, A 0, B 90, C -0, E1 0, E2 0, E3 0, E4 0} C_DIS
LIN {X 781.237, Y -399.909, Z 112.8, A 0, B 90, C -0, E1 0, E2 0, E3 0, E4 0} C_DIS
LIN {X 781.121, Y -398.789, Z 112.8, A 0, B 90, C -0, E1 0, E2 0, E3 0, E4 0} C_DIS
LIN {X 781.74, Y -393.11, Z 112.8, A 0, B 90, C -0, E1 0, E2 0, E3 0, E4 0} C_DIS
LIN {X 781.498, Y -392.042, Z 112.8, A 0, B 90, C -0, E1 0, E2 0, E3 0, E4 0} C_DIS
LIN {X 780.406, Y -391.821, Z 112.8, A 0, B 90, C -0, E1 0, E2 0, E3 0, E4 0} C_DIS
LIN {X 774.695, Y -391.937, Z 112.8, A 0, B 90, C -0, E1 0, E2 0, E3 0, E4 0} C_DIS
LIN {X 773.613, Y -391.639, Z 112.8, A 0, B 90, C -0, E1 0, E2 0, E3 0, E4 0} C_DIS
LIN {X 772.953, Y -390.726, Z 112.8, A 0, B 90, C -0, E1 0, E2 0, E3 0, E4 0} C_DIS
LIN {X 770.649, Y -385.499, Z 112.8, A 0, B 90, C -0, E1 0, E2 0, E3 0, E4 0} C_DIS
LIN {X 769.906, Y -384.696, Z 112.8, A 0, B 90, C -0, E1 0, E2 0, E3 0, E4 0} C_DIS
LIN {X 768.85, Y -385.05, Z 112.8, A 0, B 90, C -0, E1 0, E2 0, E3 0, E4 0} C_DIS
LIN {X 764.939, Y -387.415, Z 112.8, A 0, B 90, C -0, E1 0, E2 0, E3 0, E4 0} C_DIS
LIN {X 763.8, Y -388.069, Z 113.45, A 0, B 90, C -0, E1 0, E2 0, E3 0, E4 0} C_DIS
LIN {X 762.719, Y -388.359, Z 113.45, A 0, B 90, C -0, E1 0, E2 0, E3 0, E4 0} C_DIS
LIN {X 761.692, Y -387.908, Z 113.45, A 0, B 90, C -0, E1 0, E2 0, E3 0, E4 0} C_DIS
LIN {X 757.076, Y -384.577, Z 113.45, A 0, B 90, C -0, E1 0, E2 0, E3 0, E4 0} C_DIS
LIN {X 756.031, Y -384.261, Z 113.45, A 0, B 90, C -0, E1 0, E2 0, E3 0, E4 0} C_DIS
LIN {X 755.303, Y -385.099, Z 113.45, A 0, B 90, C -0, E1 0, E2 0, E3 0, E4 0} C_DIS
LIN {X 752.592, Y -390.104, Z 113.45, A 0, B 90, C -0, E1 0, E2 0, E3 0, E4 0} C_DIS
LIN {X 751.801, Y -390.895, Z 113.45, A 0, B 90, C -0, E1 0, E2 0, E3 0, E4 0} C_DIS
LIN {X 750.686, Y -391.018, Z 113.45, A 0, B 90, C -0, E1 0, E2 0, E3 0, E4 0} C_DIS
LIN {X 745.023, Y -390.441, Z 113.45, A 0, B 90, C -0, E1 0, E2 0, E3 0, E4 0} C_DIS
LIN {X 743.961, Y -390.69, Z 113.45, A 0, B 90, C -0, E1 0, E2 0, E3 0, E4 0} C_DIS
LIN {X 743.748, Y -391.78, Z 113.45, A 0, B 90, C -0, E1 0, E2 0, E3 0, E4 0} C_DIS
LIN {X 743.904, Y -397.469, Z 113.45, A 0, B 90, C -0, E1 0, E2 0, E3 0, E4 0} C_DIS
LIN {X 743.614, Y -398.55, Z 113.45, A 0, B 90, C -0, E1 0, E2 0, E3 0, E4 0} C_DIS
LIN {X 742.709, Y -399.214, Z 113.45, A 0, B 90, C -0, E1 0, E2 0, E3 0, E4 0} C_DIS
LIN {X 737.517, Y -401.546, Z 113.45, A 0, B 90, C -0, E1 0, E2 0, E3 0, E4 0} C_DIS
LIN {X 736.722, Y -402.293, Z 113.45, A 0, B 90, C -0, E1 0, E2 0, E3 0, E4 0} C_DIS
LIN {X 737.082, Y -403.343, Z 113.45, A 0, B 90, C -0, E1 0, E2 0, E3 0, E4 0} C_DIS
LIN {X 740.062, Y -408.193, Z 113.45, A 0, B 90, C -0, E1 0, E2 0, E3 0, E4 0} C_DIS
LIN {X 740.351, Y -409.273, Z 113.45, A 0, B 90, C -0, E1 0, E2 0, E3 0, E4 0} C_DIS
LIN {X 739.9, Y -410.301, Z 113.45, A 0, B 90, C -0, E1 0, E2 0, E3 0, E4 0} C_DIS
LIN {X 736.569, Y -414.916, Z 113.45, A 0, B 90, C -0, E1 0, E2 0, E3 0, E4 0} C_DIS
LIN {X 736.254, Y -415.961, Z 113.45, A 0, B 90, C -0, E1 0, E2 0, E3 0, E4 0} C_DIS
LIN {X 737.091, Y -416.69, Z 113.45, A 0, B 90, C -0, E1 0, E2 0, E3 0, E4 0} C_DIS
LIN {X 742.096, Y -419.4, Z 113.45, A 0, B 90, C -0, E1 0, E2 0, E3 0, E4 0} C_DIS
LIN {X 742.887, Y -420.191, Z 113.45, A 0, B 90, C -0, E1 0, E2 0, E3 0, E4 0} C_DIS
LIN {X 743.01, Y -421.307, Z 113.45, A 0, B 90, C -0, E1 0, E2 0, E3 0, E4 0} C_DIS
LIN {X 742.434, Y -426.969, Z 113.45, A 0, B 90, C -0, E1 0, E2 0, E3 0, E4 0} C_DIS
LIN {X 742.683, Y -428.032, Z 113.45, A 0, B 90, C -0, E1 0, E2 0, E3 0, E4 0} C_DIS
LIN {X 743.772, Y -428.244, Z 113.45, A 0, B 90, C -0, E1 0, E2 0, E3 0, E4 0} C_DIS
LIN {X 749.462, Y -428.089, Z 113.45, A 0, B 90, C -0, E1 0, E2 0, E3 0, E4 0} C_DIS
LIN {X 750.542, Y -428.378, Z 113.45, A 0, B 90, C -0, E1 0, E2 0, E3 0, E4 0} C_DIS
LIN {X 751.207, Y -429.283, Z 113.45, A 0, B 90, C -0, E1 0, E2 0, E3 0, E4 0} C_DIS
LIN {X 753.539, Y -434.475, Z 113.45, A 0, B 90, C -0, E1 0, E2 0, E3 0, E4 0} C_DIS
LIN {X 754.286, Y -435.271, Z 113.45, A 0, B 90, C -0, E1 0, E2 0, E3 0, E4 0} C_DIS
LIN {X 755.335, Y -434.91, Z 113.45, A 0, B 90, C -0, E1 0, E2 0, E3 0, E4 0} C_DIS
LIN {X 760.185, Y -431.931, Z 113.45, A 0, B 90, C -0, E1 0, E2 0, E3 0, E4 0} C_DIS
LIN {X 761.266, Y -431.641, Z 113.45, A 0, B 90, C -0, E1 0, E2 0, E3 0, E4 0} C_DIS
LIN {X 762.293, Y -432.092, Z 113.45, A 0, B 90, C -0, E1 0, E2 0, E3 0, E4 0} C_DIS
LIN {X 766.909, Y -435.423, Z 113.45, A 0, B 90, C -0, E1 0, E2 0, E3 0, E4 0} C_DIS
LIN {X 767.954, Y -435.739, Z 113.45, A 0, B 90, C -0, E1 0, E2 0, E3 0, E4 0} C_DIS
LIN {X 768.682, Y -434.901, Z 113.45, A 0, B 90, C -0, E1 0, E2 0, E3 0, E4 0} C_DIS
LIN {X 771.393, Y -429.896, Z 113.45, A 0, B 90, C -0, E1 0, E2 0, E3 0, E4 0} C_DIS
LIN {X 772.183, Y -429.105, Z 113.45, A 0, B 90, C -0, E1 0, E2 0, E3 0, E4 0} C_DIS
LIN {X 773.299, Y -428.982, Z 113.45, A 0, B 90, C -0, E1 0, E2 0, E3 0, E4 0} C_DIS
LIN {X 778.962, Y -429.559, Z 113.45, A 0, B 90, C -0, E1 0, E2 0, E3 0, E4 0} C_DIS
LIN {X 780.024, Y -429.31, Z 113.45, A 0, B 90, C -0, E1 0, E2 0, E3 0, E4 0} C_DIS
LIN {X 780.237, Y -428.22, Z 113.45, A 0, B 90, C -0, E1 0, E2 0, E3 0, E4 0} C_DIS
LIN {X 780.081, Y -422.531, Z 113.45, A 0, B 90, C -0, E1 0, E2 0, E3 0, E4 0} C_DIS
LIN {X 780.371, Y -421.45, Z 113.45, A 0, B 90, C -0, E1 0, E2 0, E3 0, E4 0} C_DIS
LIN {X 781.276, Y -420.786, Z 113.45, A 0, B 90, C -0, E1 0, E2 0, E3 0, E4 0} C_DIS
LIN {X 786.468, Y -418.454, Z 113.45, A 0, B 90, C -0, E1 0, E2 0, E3 0, E4 0} C_DIS
LIN {X 787.263, Y -417.707, Z 113.45, A 0, B 90, C -0, E1 0, E2 0, E3 0, E4 0} C_DIS
LIN {X 786.903, Y -416.657, Z 113.45, A 0, B 90, C -0, E1 0, E2 0, E3 0, E4 0} C_DIS
LIN {X 783.923, Y -411.807, Z 113.45, A 0, B 90, C -0, E1 0, E2 0, E3 0, E4 0} C_DIS
LIN {X 783.634, Y -410.727, Z 113.45, A 0, B 90, C -0, E1 0, E2 0, E3 0, E4 0} C_DIS
LIN {X 784.085, Y -409.699, Z 113.45, A 0, B 90, C -0, E1 0, E2 0, E3 0, E4 0} C_DIS
LIN {X 787.416, Y -405.084, Z 113.45, A 0, B 90, C -0, E1 0, E2 0, E3 0, E4 0} C_DIS
LIN {X 787.731, Y -404.039, Z 113.45, A 0, B 90, C -0, E1 0, E2 0, E3 0, E4 0} C_DIS
LIN {X 786.894, Y -403.31, Z 113.45, A 0, B 90, C -0, E1 0, E2 0, E3 0, E4 0} C_DIS
LIN {X 781.889, Y -400.6, Z 113.45, A 0, B 90, C -0, E1 0, E2 0, E3 0, E4 0} C_DIS
LIN {X 781.098, Y -399.809, Z 113.45, A 0, B 90, C -0, E1 0, E2 0, E3 0, E4 0} C_DIS
LIN {X 780.975, Y -398.693, Z 113.45, A 0, B 90, C -0, E1 0, E2 0, E3 0, E4 0} C_DIS
LIN {X 781.551, Y -393.031, Z 113.45, A 0, B 90, C -0, E1 0, E2 0, E3 0, E4 0} C_DIS
LIN {X 781.302, Y -391.968, Z 113.45, A 0, B 90, C -0, E1 0, E2 0, E3 0, E4 0} C_DIS
LIN {X 780.213, Y -391.756, Z 113.45, A 0, B 90, C -0, E1 0, E2 0, E3 0, E4 0} C_DIS
LIN {X 774.523, Y -391.911, Z 113.45, A 0, B 90, C -0, E1 0, E2 0, E3 0, E4 0} C_DIS
LIN {X 773.443, Y -391.622, Z 113.45, A 0, B 90, C -0, E1 0, E2 0, E3 0, E4 0} C_DIS
LIN {X 772.778, Y -390.717, Z 113.45, A 0, B 90, C -0, E1 0, E2 0, E3 0, E4 0} C_DIS
LIN {X 770.446, Y -385.525, Z 113.45, A 0, B 90, C -0, E1 0, E2 0, E3 0, E4 0} C_DIS
LIN {X 769.699, Y -384.729, Z 113.45, A 0, B 90, C -0, E1 0, E2 0, E3 0, E4 0} C_DIS
LIN {X 768.65, Y -385.09, Z 113.45, A 0, B 90, C -0, E1 0, E2 0, E3 0, E4 0} C_DIS
LIN {X 764.77, Y -387.474, Z 113.45, A 0, B 90, C -0, E1 0, E2 0, E3 0, E4 0} C_DIS
LIN {X 763.64, Y -388.133, Z 114.1, A 0, B 90, C -0, E1 0, E2 0, E3 0, E4 0} C_DIS
LIN {X 762.566, Y -388.429, Z 114.1, A 0, B 90, C -0, E1 0, E2 0, E3 0, E4 0} C_DIS
LIN {X 761.538, Y -387.986, Z 114.1, A 0, B 90, C -0, E1 0, E2 0, E3 0, E4 0} C_DIS
LIN {X 756.915, Y -384.7, Z 114.1, A 0, B 90, C -0, E1 0, E2 0, E3 0, E4 0} C_DIS
LIN {X 755.872, Y -384.392, Z 114.1, A 0, B 90, C -0, E1 0, E2 0, E3 0, E4 0} C_DIS
LIN {X 755.152, Y -385.232, Z 114.1, A 0, B 90, C -0, E1 0, E2 0, E3 0, E4 0} C_DIS
LIN {X 752.486, Y -390.239, Z 114.1, A 0, B 90, C -0, E1 0, E2 0, E3 0, E4 0} C_DIS
LIN {X 751.703, Y -391.032, Z 114.1, A 0, B 90, C -0, E1 0, E2 0, E3 0, E4 0} C_DIS
LIN {X 750.592, Y -391.163, Z 114.1, A 0, B 90, C -0, E1 0, E2 0, E3 0, E4 0} C_DIS
LIN {X 744.945, Y -390.628, Z 114.1, A 0, B 90, C -0, E1 0, E2 0, E3 0, E4 0} C_DIS
LIN {X 743.888, Y -390.883, Z 114.1, A 0, B 90, C -0, E1 0, E2 0, E3 0, E4 0} C_DIS
LIN {X 743.684, Y -391.97, Z 114.1, A 0, B 90, C -0, E1 0, E2 0, E3 0, E4 0} C_DIS
LIN {X 743.879, Y -397.639, Z 114.1, A 0, B 90, C -0, E1 0, E2 0, E3 0, E4 0} C_DIS
LIN {X 743.598, Y -398.718, Z 114.1, A 0, B 90, C -0, E1 0, E2 0, E3 0, E4 0} C_DIS
LIN {X 742.701, Y -399.386, Z 114.1, A 0, B 90, C -0, E1 0, E2 0, E3 0, E4 0} C_DIS
LIN {X 737.543, Y -401.747, Z 114.1, A 0, B 90, C -0, E1 0, E2 0, E3 0, E4 0} C_DIS
LIN {X 736.755, Y -402.497, Z 114.1, A 0, B 90, C -0, E1 0, E2 0, E3 0, E4 0} C_DIS
LIN {X 737.122, Y -403.54, Z 114.1, A 0, B 90, C -0, E1 0, E2 0, E3 0, E4 0} C_DIS
LIN {X 740.125, Y -408.352, Z 114.1, A 0, B 90, C -0, E1 0, E2 0, E3 0, E4 0} C_DIS
LIN {X 740.421, Y -409.427, Z 114.1, A 0, B 90, C -0, E1 0, E2 0, E3 0, E4 0} C_DIS
LIN {X 739.979, Y -410.454, Z 114.1, A 0, B 90, C -0, E1 0, E2 0, E3 0, E4 0} C_DIS
LIN {X 736.692, Y -415.077, Z 114.1, A 0, B 90, C -0, E1 0, E2 0, E3 0, E4 0} C_DIS
LIN {X 736.385, Y -416.12, Z 114.1, A 0, B 90, C -0, E1 0, E2 0, E3 0, E4 0} C_DIS
LIN {X 737.224, Y -416.841, Z 114.1, A 0, B 90, C -0, E1 0, E2 0, E3 0, E4 0} C_DIS
LIN {X 742.231, Y -419.507, Z 114.1, A 0, B 90, C -0, E1 0, E2 0, E3 0, E4 0} C_DIS
LIN {X 743.025, Y -420.289, Z 114.1, A 0, B 90, C -0, E1 0, E2 0, E3 0, E4 0} C_DIS
LIN {X 743.155, Y -421.4, Z 114.1, A 0, B 90, C -0, E1 0, E2 0, E3 0, E4 0} C_DIS
LIN {X 742.62, Y -427.047, Z 114.1, A 0, B 90, C -0, E1 0, E2 0, E3 0, E4 0} C_DIS
LIN {X 742.876, Y -428.104, Z 114.1, A 0, B 90, C -0, E1 0, E2 0, E3 0, E4 0} C_DIS
LIN {X 743.963, Y -428.308, Z 114.1, A 0, B 90, C -0, E1 0, E2 0, E3 0, E4 0} C_DIS
LIN {X 749.632, Y -428.114, Z 114.1, A 0, B 90, C -0, E1 0, E2 0, E3 0, E4 0} C_DIS
LIN {X 750.711, Y -428.395, Z 114.1, A 0, B 90, C -0, E1 0, E2 0, E3 0, E4 0} C_DIS
LIN {X 751.379, Y -429.292, Z 114.1, A 0, B 90, C -0, E1 0, E2 0, E3 0, E4 0} C_DIS
LIN {X 753.739, Y -434.449, Z 114.1, A 0, B 90, C -0, E1 0, E2 0, E3 0, E4 0} C_DIS
LIN {X 754.489, Y -435.237, Z 114.1, A 0, B 90, C -0, E1 0, E2 0, E3 0, E4 0} C_DIS
LIN {X 755.533, Y -434.87, Z 114.1, A 0, B 90, C -0, E1 0, E2 0, E3 0, E4 0} C_DIS
LIN {X 760.345, Y -431.867, Z 114.1, A 0, B 90, C -0, E1 0, E2 0, E3 0, E4 0} C_DIS
LIN {X 761.419, Y -431.571, Z 114.1, A 0, B 90, C -0, E1 0, E2 0, E3 0, E4 0} C_DIS
LIN {X 762.447, Y -432.014, Z 114.1, A 0, B 90, C -0, E1 0, E2 0, E3 0, E4 0} C_DIS
LIN {X 767.07, Y -435.3, Z 114.1, A 0, B 90, C -0, E1 0, E2 0, E3 0, E4 0} C_DIS
LIN {X 768.113, Y -435.608, Z 114.1, A 0, B 90, C -0, E1 0, E2 0, E3 0, E4 0} C_DIS
LIN {X 768.833, Y -434.768, Z 114.1, A 0, B 90, C -0, E1 0, E2 0, E3 0, E4 0} C_DIS
LIN {X 771.499, Y -429.761, Z 114.1, A 0, B 90, C -0, E1 0, E2 0, E3 0, E4 0} C_DIS
LIN {X 772.282, Y -428.968, Z 114.1, A 0, B 90, C -0, E1 0, E2 0, E3 0, E4 0} C_DIS
LIN {X 773.393, Y -428.837, Z 114.1, A 0, B 90, C -0, E1 0, E2 0, E3 0, E4 0} C_DIS
LIN {X 779.04, Y -429.372, Z 114.1, A 0, B 90, C -0, E1 0, E2 0, E3 0, E4 0} C_DIS
LIN {X 780.097, Y -429.117, Z 114.1, A 0, B 90, C -0, E1 0, E2 0, E3 0, E4 0} C_DIS
LIN {X 780.301, Y -428.03, Z 114.1, A 0, B 90, C -0, E1 0, E2 0, E3 0, E4 0} C_DIS
LIN {X 780.106, Y -422.361, Z 114.1, A 0, B 90, C -0, E1 0, E2 0, E3 0, E4 0} C_DIS
LIN {X 780.387, Y -421.282, Z 114.1, A 0, B 90, C -0, E1 0, E2 0, E3 0, E4 0} C_DIS
LIN {X 781.284, Y -420.614, Z 114.1, A 0, B 90, C -0, E1 0, E2 0, E3 0, E4 0} C_DIS
LIN {X 786.442, Y -418.253, Z 114.1, A 0, B 90, C -0, E1 0, E2 0, E3 0, E4 0} C_DIS
LIN {X 787.23, Y -417.503, Z 114.1, A 0, B 90, C -0, E1 0, E2 0, E3 0, E4 0} C_DIS
LIN {X 786.863, Y -416.46, Z 114.1, A 0, B 90, C -0, E1 0, E2 0, E3 0, E4 0} C_DIS
LIN {X 783.86, Y -411.648, Z 114.1, A 0, B 90, C -0, E1 0, E2 0, E3 0, E4 0} C_DIS
LIN {X 783.564, Y -410.573, Z 114.1, A 0, B 90, C -0, E1 0, E2 0, E3 0, E4 0} C_DIS
LIN {X 784.006, Y -409.546, Z 114.1, A 0, B 90, C -0, E1 0, E2 0, E3 0, E4 0} C_DIS
LIN {X 787.293, Y -404.923, Z 114.1, A 0, B 90, C -0, E1 0, E2 0, E3 0, E4 0} C_DIS
LIN {X 787.6, Y -403.88, Z 114.1, A 0, B 90, C -0, E1 0, E2 0, E3 0, E4 0} C_DIS
LIN {X 786.761, Y -403.159, Z 114.1, A 0, B 90, C -0, E1 0, E2 0, E3 0, E4 0} C_DIS
LIN {X 781.754, Y -400.493, Z 114.1, A 0, B 90, C -0, E1 0, E2 0, E3 0, E4 0} C_DIS
LIN {X 780.96, Y -399.711, Z 114.1, A 0, B 90, C -0, E1 0, E2 0, E3 0, E4 0} C_DIS
LIN {X 780.83, Y -398.6, Z 114.1, A 0, B 90, C -0, E1 0, E2 0, E3 0, E4 0} C_DIS
LIN {X 781.365, Y -392.953, Z 114.1, A 0, B 90, C -0, E1 0, E2 0, E3 0, E4 0} C_DIS
LIN {X 781.109, Y -391.896, Z 114.1, A 0, B 90, C -0, E1 0, E2 0, E3 0, E4 0} C_DIS
LIN {X 780.022, Y -391.692, Z 114.1, A 0, B 90, C -0, E1 0, E2 0, E3 0, E4 0} C_DIS
LIN {X 774.353, Y -391.886, Z 114.1, A 0, B 90, C -0, E1 0, E2 0, E3 0, E4 0} C_DIS
LIN {X 773.274, Y -391.605, Z 114.1, A 0, B 90, C -0, E1 0, E2 0, E3 0, E4 0} C_DIS
LIN {X 772.606, Y -390.708, Z 114.1, A 0, B 90, C -0, E1 0, E2 0, E3 0, E4 0} C_DIS
LIN {X 770.246, Y -385.551, Z 114.1, A 0, B 90, C -0, E1 0, E2 0, E3 0, E4 0} C_DIS
LIN {X 769.496, Y -384.763, Z 114.1, A 0, B 90, C -0, E1 0, E2 0, E3 0, E4 0} C_DIS
LIN {X 768.452, Y -385.13, Z 114.1, A 0, B 90, C -0, E1 0, E2 0, E3 0, E4 0} C_DIS
LIN {X 764.603, Y -387.532, Z 114.1, A 0, B 90, C -0, E1 0, E2 0, E3 0, E4 0} C_DIS
LIN {X 763.483, Y -388.196, Z 114.75, A 0, B 90, C -0, E1 0, E2 0, E3 0, E4 0} C_DIS
LIN {X 762.414, Y -388.499, Z 114.75, A 0, B 90, C -0, E1 0, E2 0, E3 0, E4 0} C_DIS
LIN {X 761.387, Y -388.065, Z 114.75, A 0, B 90, C -0, E1 0, E2 0, E3 0, E4 0} C_DIS
LIN {X 756.757, Y -384.821, Z 114.75, A 0, B 90, C -0, E1 0, E2 0, E3 0, E4 0} C_DIS
LIN {X 755.715, Y -384.522, Z 114.75, A 0, B 90, C -0, E1 0, E2 0, E3 0, E4 0} C_DIS
LIN {X 755.003, Y -385.364, Z 114.75, A 0, B 90, C -0, E1 0, E2 0, E3 0, E4 0} C_DIS
LIN {X 752.381, Y -390.372, Z 114.75, A 0, B 90, C -0, E1 0, E2 0, E3 0, E4 0} C_DIS
LIN {X 751.607, Y -391.168, Z 114.75, A 0, B 90, C -0, E1 0, E2 0, E3 0, E4 0} C_DIS
LIN {X 750.501, Y -391.306, Z 114.75, A 0, B 90, C -0, E1 0, E2 0, E3 0, E4 0} C_DIS
LIN {X 744.869, Y -390.812, Z 114.75, A 0, B 90, C -0, E1 0, E2 0, E3 0, E4 0} C_DIS
LIN {X 743.818, Y -391.074, Z 114.75, A 0, B 90, C -0, E1 0, E2 0, E3 0, E4 0} C_DIS
LIN {X 743.622, Y -392.159, Z 114.75, A 0, B 90, C -0, E1 0, E2 0, E3 0, E4 0} C_DIS
LIN {X 743.855, Y -397.807, Z 114.75, A 0, B 90, C -0, E1 0, E2 0, E3 0, E4 0} C_DIS
LIN {X 743.583, Y -398.884, Z 114.75, A 0, B 90, C -0, E1 0, E2 0, E3 0, E4 0} C_DIS
LIN {X 742.693, Y -399.556, Z 114.75, A 0, B 90, C -0, E1 0, E2 0, E3 0, E4 0} C_DIS
LIN {X 737.569, Y -401.944, Z 114.75, A 0, B 90, C -0, E1 0, E2 0, E3 0, E4 0} C_DIS
LIN {X 736.789, Y -402.697, Z 114.75, A 0, B 90, C -0, E1 0, E2 0, E3 0, E4 0} C_DIS
LIN {X 737.162, Y -403.735, Z 114.75, A 0, B 90, C -0, E1 0, E2 0, E3 0, E4 0} C_DIS
LIN {X 740.189, Y -408.509, Z 114.75, A 0, B 90, C -0, E1 0, E2 0, E3 0, E4 0} C_DIS
LIN {X 740.491, Y -409.578, Z 114.75, A 0, B 90, C -0, E1 0, E2 0, E3 0, E4 0} C_DIS
LIN {X 740.057, Y -410.605, Z 114.75, A 0, B 90, C -0, E1 0, E2 0, E3 0, E4 0} C_DIS
LIN {X 736.814, Y -415.235, Z 114.75, A 0, B 90, C -0, E1 0, E2 0, E3 0, E4 0} C_DIS
LIN {X 736.515, Y -416.277, Z 114.75, A 0, B 90, C -0, E1 0, E2 0, E3 0, E4 0} C_DIS
LIN {X 737.356, Y -416.989, Z 114.75, A 0, B 90, C -0, E1 0, E2 0, E3 0, E4 0} C_DIS
LIN {X 742.365, Y -419.611, Z 114.75, A 0, B 90, C -0, E1 0, E2 0, E3 0, E4 0} C_DIS
LIN {X 743.161, Y -420.386, Z 114.75, A 0, B 90, C -0, E1 0, E2 0, E3 0, E4 0} C_DIS
LIN {X 743.298, Y -421.492, Z 114.75, A 0, B 90, C -0, E1 0, E2 0, E3 0, E4 0} C_DIS
LIN {X 742.805, Y -427.123, Z 114.75, A 0, B 90, C -0, E1 0, E2 0, E3 0, E4 0} C_DIS
LIN {X 743.067, Y -428.175, Z 114.75, A 0, B 90, C -0, E1 0, E2 0, E3 0, E4 0} C_DIS
LIN {X 744.151, Y -428.371, Z 114.75, A 0, B 90, C -0, E1 0, E2 0, E3 0, E4 0} C_DIS
LIN {X 749.8, Y -428.137, Z 114.75, A 0, B 90, C -0, E1 0, E2 0, E3 0, E4 0} C_DIS
LIN {X 750.877, Y -428.41, Z 114.75, A 0, B 90, C -0, E1 0, E2 0, E3 0, E4 0} C_DIS
LIN {X 751.549, Y -429.299, Z 114.75, A 0, B 90, C -0, E1 0, E2 0, E3 0, E4 0} C_DIS
LIN {X 753.937, Y -434.423, Z 114.75, A 0, B 90, C -0, E1 0, E2 0, E3 0, E4 0} C_DIS
LIN {X 754.69, Y -435.203, Z 114.75, A 0, B 90, C -0, E1 0, E2 0, E3 0, E4 0} C_DIS
LIN {X 755.727, Y -434.83, Z 114.75, A 0, B 90, C -0, E1 0, E2 0, E3 0, E4 0} C_DIS
LIN {X 760.502, Y -431.804, Z 114.75, A 0, B 90, C -0, E1 0, E2 0, E3 0, E4 0} C_DIS
LIN {X 761.571, Y -431.501, Z 114.75, A 0, B 90, C -0, E1 0, E2 0, E3 0, E4 0} C_DIS
LIN {X 762.598, Y -431.935, Z 114.75, A 0, B 90, C -0, E1 0, E2 0, E3 0, E4 0} C_DIS
LIN {X 767.228, Y -435.179, Z 114.75, A 0, B 90, C -0, E1 0, E2 0, E3 0, E4 0} C_DIS
LIN {X 768.269, Y -435.478, Z 114.75, A 0, B 90, C -0, E1 0, E2 0, E3 0, E4 0} C_DIS
LIN {X 768.982, Y -434.636, Z 114.75, A 0, B 90, C -0, E1 0, E2 0, E3 0, E4 0} C_DIS
LIN {X 771.604, Y -429.628, Z 114.75, A 0, B 90, C -0, E1 0, E2 0, E3 0, E4 0} C_DIS
LIN {X 772.378, Y -428.832, Z 114.75, A 0, B 90, C -0, E1 0, E2 0, E3 0, E4 0} C_DIS
LIN {X 773.484, Y -428.694, Z 114.75, A 0, B 90, C -0, E1 0, E2 0, E3 0, E4 0} C_DIS
LIN {X 779.116, Y -429.188, Z 114.75, A 0, B 90, C -0, E1 0, E2 0, E3 0, E4 0} C_DIS
LIN {X 780.167, Y -428.926, Z 114.75, A 0, B 90, C -0, E1 0, E2 0, E3 0, E4 0} C_DIS
LIN {X 780.363, Y -427.841, Z 114.75, A 0, B 90, C -0, E1 0, E2 0, E3 0, E4 0} C_DIS
LIN {X 780.13, Y -422.193, Z 114.75, A 0, B 90, C -0, E1 0, E2 0, E3 0, E4 0} C_DIS
LIN {X 780.402, Y -421.116, Z 114.75, A 0, B 90, C -0, E1 0, E2 0, E3 0, E4 0} C_DIS
LIN {X 781.292, Y -420.444, Z 114.75, A 0, B 90, C -0, E1 0, E2 0, E3 0, E4 0} C_DIS
LIN {X 786.416, Y -418.056, Z 114.75, A 0, B 90, C -0, E1 0, E2 0, E3 0, E4 0} C_DIS
LIN {X 787.195, Y -417.303, Z 114.75, A 0, B 90, C -0, E1 0, E2 0, E3 0, E4 0} C_DIS
LIN {X 786.823, Y -416.265, Z 114.75, A 0, B 90, C -0, E1 0, E2 0, E3 0, E4 0} C_DIS
LIN {X 783.796, Y -411.491, Z 114.75, A 0, B 90, C -0, E1 0, E2 0, E3 0, E4 0} C_DIS
LIN {X 783.494, Y -410.422, Z 114.75, A 0, B 90, C -0, E1 0, E2 0, E3 0, E4 0} C_DIS
LIN {X 783.928, Y -409.395, Z 114.75, A 0, B 90, C -0, E1 0, E2 0, E3 0, E4 0} C_DIS
LIN {X 787.171, Y -404.765, Z 114.75, A 0, B 90, C -0, E1 0, E2 0, E3 0, E4 0} C_DIS
LIN {X 787.47, Y -403.723, Z 114.75, A 0, B 90, C -0, E1 0, E2 0, E3 0, E4 0} C_DIS
LIN {X 786.629, Y -403.011, Z 114.75, A 0, B 90, C -0, E1 0, E2 0, E3 0, E4 0} C_DIS
LIN {X 781.62, Y -400.389, Z 114.75, A 0, B 90, C -0, E1 0, E2 0, E3 0, E4 0} C_DIS
LIN {X 780.824, Y -399.614, Z 114.75, A 0, B 90, C -0, E1 0, E2 0, E3 0, E4 0} C_DIS
LIN {X 780.686, Y -398.508, Z 114.75, A 0, B 90, C -0, E1 0, E2 0, E3 0, E4 0} C_DIS
LIN {X 781.18, Y -392.877, Z 114.75, A 0, B 90, C -0, E1 0, E2 0, E3 0, E4 0} C_DIS
LIN {X 780.918, Y -391.825, Z 114.75, A 0, B 90, C -0, E1 0, E2 0, E3 0, E4 0} C_DIS
LIN {X 779.833, Y -391.629, Z 114.75, A 0, B 90, C -0, E1 0, E2 0, E3 0, E4 0} C_DIS
LIN {X 774.185, Y -391.863, Z 114.75, A 0, B 90, C -0, E1 0, E2 0, E3 0, E4 0} C_DIS
LIN {X 773.108, Y -391.59, Z 114.75, A 0, B 90, C -0, E1 0, E2 0, E3 0, E4 0} C_DIS
LIN {X 772.436, Y -390.701, Z 114.75, A 0, B 90, C -0, E1 0, E2 0, E3 0, E4 0} C_DIS
LIN {X 770.048, Y -385.577, Z 114.75, A 0, B 90, C -0, E1 0, E2 0, E3 0, E4 0} C_DIS
LIN {X 769.295, Y -384.797, Z 114.75, A 0, B 90, C -0, E1 0, E2 0, E3 0, E4 0} C_DIS
LIN {X 768.258, Y -385.17, Z 114.75, A 0, B 90, C -0, E1 0, E2 0, E3 0, E4 0} C_DIS
LIN {X 764.438, Y -387.591, Z 114.75, A 0, B 90, C -0, E1 0, E2 0, E3 0, E4 0} C_DIS
LIN {X 763.328, Y -388.259, Z 115.4, A 0, B 90, C -0, E1 0, E2 0, E3 0, E4 0} C_DIS
LIN {X 762.265, Y -388.568, Z 115.4, A 0, B 90, C -0, E1 0, E2 0, E3 0, E4 0} C_DIS
LIN {X 761.238, Y -388.142, Z 115.4, A 0, B 90, C -0, E1 0, E2 0, E3 0, E4 0} C_DIS
LIN {X 756.602, Y -384.942, Z 115.4, A 0, B 90, C -0, E1 0, E2 0, E3 0, E4 0} C_DIS
LIN {X 755.561, Y -384.651, Z 115.4, A 0, B 90, C -0, E1 0, E2 0, E3 0, E4 0} C_DIS
LIN {X 754.857, Y -385.495, Z 115.4, A 0, B 90, C -0, E1 0, E2 0, E3 0, E4 0} C_DIS
LIN {X 752.279, Y -390.504, Z 115.4, A 0, B 90, C -0, E1 0, E2 0, E3 0, E4 0} C_DIS
LIN {X 751.512, Y -391.303, Z 115.4, A 0, B 90, C -0, E1 0, E2 0, E3 0, E4 0} C_DIS
LIN {X 750.411, Y -391.448, Z 115.4, A 0, B 90, C -0, E1 0, E2 0, E3 0, E4 0} C_DIS
